// ---- 11_CNC/01_DUTs/02_ST/ST_CNC_Heidenhain_Exchange_Out_1.TcDUT
//-----------------------------------------------------------------------------------------
//
//                  				ST_CNC_Heidenhain_Exchange_Out
//
//								Structure Echange Magasin->CNC_Heidenhain 			
//-----------------------------------------------------------------------------------------
//
//Auteur: G.GOETZ (In agreement with ...)
//Création: 27.01.2026
//Dernière modification : 27.01.2026 (G.GOETZ)
//       			
//-----------------------------------------------------------------------------------------
//
//     							Liste des modifications  	
//
// 27.01.2026 (G.GOETZ) -> Création		
//-----------------------------------------------------------------------------------------

TYPE ST_CNC_Heidenhain_Exchange_Out_1 : // 16 Bytes -> Start at X0.0 / End at X15.7 (X0.0+15.7)
STRUCT
	
	(* Byte 0 *)
		boLife : BIT ; // Magazine Life bit -> X0.0
		boReserve01 : BIT ; // Reserve 01 -> X0.1
		boReserve02 : BIT ; // Reserve 02 -> X0.2
		boReserve03 : BIT ; // Reserve 03 -> X0.3
		boReserve04 : BIT ; // Reserve 04 -> X0.4
		boReserve05 : BIT ; // Reserve 05 -> X0.5
		boLoadingArmInPosition : BIT ; // Loading Arm in position in the CNC -> X0.6
		boNoFault : BIT ; // No Fault on the Magazine -> X0.7

	(* Byte 1 *)
		boReserve10 : BIT ; // Reserve 10 -> X1.0
		boReserve11 : BIT ; // Reserve 11 -> X1.1
		boReserve12 : BIT ; // Reserve 12 -> X1.2
		boReserve13 : BIT ; // Reserve 13 -> X1.3
		boReserve14 : BIT ; // Reserve 14 -> X1.4
		boReserve15 : BIT ; // Reserve 15 -> X1.5
		boReserve16 : BIT ; // Reserve 16 -> X1.6
		boDoorClosed : BIT ; // Magazine Door closed (operator) -> X1.7

	(* Byte 2 *)
		boReserve20 : BIT ; // Reserve 20 -> X2.0
		boReserve21 : BIT ; // Reserve 21 -> X2.1
		boReserve22 : BIT ; // Reserve 22 -> X2.2
		boReserve23 : BIT ; // Reserve 23 -> X2.3
		boReserve24 : BIT ; // Reserve 24 -> X2.4
		boReserve25 : BIT ; // Reserve 25 -> X2.5
		boReserve26 : BIT ; // Reserve 26 -> X2.6
		boReserve27 : BIT ; // Reserve 27 -> X2.7
	
	(* Byte 3 *)
		boReserve30 : BIT ; // Reserve 30 -> X3.0
		boReserve31 : BIT ; // Reserve 31 -> X3.1
		boReserve32 : BIT ; // Reserve 32 -> X3.2
		boReserve33 : BIT ; // Reserve 33 -> X3.3
		boReserve34 : BIT ; // Reserve 34 -> X3.4
		boReserve35 : BIT ; // Reserve 35 -> X3.5
		boReserve36 : BIT ; // Reserve 36 -> X3.6
		boReserve37 : BIT ; // Reserve 37 -> X3.7

	(* Byte 4 *)
		byoReserve40 : BYTE ; // Reserve 40 -> X4
	
	(* Byte 5 *)
		byoReserve50 : BYTE ; // Reserve 50 -> X5
	
	(* Byte 6 *)
		byoReserve60 : BYTE ; // Reserve 60 -> X6
	
	(* Byte 7 *)
		byoReserve70 : BYTE ; // Reserve 70 -> X7
	
	(* Byte 8 *)
		byoReserve80 : BYTE ; // Reserve 80 -> X8
	
	(* Byte 9 *)
		byoReserve90 : BYTE ; // Reserve 90 -> X9
		
	(* Byte 10 *)
		byoReserve100 : BYTE ; // Reserve 100 -> X10
	
	(* Byte 11 *)
		byoReserve110 : BYTE ; // Reserve 110 -> X11
	
	(* Byte 12 *)
		byoReserve120 : BYTE ; // Reserve 120 -> X12
	
	(* Byte 13 *)
		byoReserve130 : BYTE ; // Reserve 130 -> X13
	
	(* Byte 14 *)
		byoReserve140 : BYTE ; // Reserve 140 -> X14
	
	(* Byte 15 *)
		byoReserve150 : BYTE ; // Reserve 150 -> X15
	
END_STRUCT
END_TYPE

// ---- 11_CNC/01_DUTs/02_ST/ST_CNC_Heidenhain_Data.TcDUT
//-----------------------------------------------------------------------------------------
//
//                  				ST_CNC_Heidenhain_Data
//
//								Structure CNC_Heidenhain Data 			
//-----------------------------------------------------------------------------------------
//
//Auteur: G.GOETZ
//Création: 27.01.2026
//Dernière modification : 27.01.2026 (G.GOETZ)
//       			
//-----------------------------------------------------------------------------------------
//
//     							Liste des modifications  	
//
// 27.01.2026 (G.GOETZ) -> Création		
//-----------------------------------------------------------------------------------------

TYPE ST_CNC_Heidenhain_Data :
STRUCT

	(** ST **)	
		stCncMagazine : ST_CNC_Heidenhain_Exchange_In_1 ; // Structure Exchange CNC -> Magazine
		stMagazineCNC : ST_CNC_Heidenhain_Exchange_Out_1 ; // Structure Exchange Magzine -> CNC

END_STRUCT
END_TYPE

// ---- 11_CNC/01_DUTs/02_ST/ST_CNC_Fanuc_Exchange_In_1.TcDUT
//-----------------------------------------------------------------------------------------
//
//                  				ST_CNC_Fanuc_Exchange_In
//
//								Structure Echange CNC_Fanuc->Magasin 			
//-----------------------------------------------------------------------------------------
//
//Auteur: G.GOETZ (In agreement with J.SPÄTIG)
//Création: 27.01.2026
//Dernière modification : 27.01.2026 (G.GOETZ)
//       			
//-----------------------------------------------------------------------------------------
//
//     							Liste des modifications  	
//
// 27.01.2026 (G.GOETZ) -> Création		
//-----------------------------------------------------------------------------------------

TYPE ST_CNC_Fanuc_Exchange_In_1 : // 32 Bytes -> Start at X0.0 / End at X31.7 (X0.0+31.7)
STRUCT
	
	(* Byte 0 *)
		byi0 AT %I* : BYTE ; // Byte X0
			biLife : BIT ; // Life bit -> X0.0
			biToolAnticipation : BIT ; // Anticipation to prepare the next Tool -> X0.1
			biAllowedOpenIntermediateDoor : BIT ; // Allowed to open the Intermediate Door 02 -> X0.2
			biLoadUnloadRequest : BIT ; // Request to Load and Unload a Tool -> X0.3
			biLoadRequest : BIT ; // Request to only Load a Tool -> X0.4
			biUnloadRequest : BIT ; // Request to only Unload a Tool -> X0.5
			biLoadUnloadEnd : BIT ; // End of the Request -> X0.6
			biAllowedCloseIntermediateDoor : BIT ; // Allowed to close the Intermediate Door 07 -> X0.7

	(* Byte 1 *)
		byi1 AT %I* : BYTE ; // Byte X1
			biInCycle : BIT ; // CNC in Cycle -> X1.0
			biEvacuateArm : BIT ; // Request to evacuate the Changing Arm and close the Intermediate Door -> X1.1
			biReserve12 : BIT ; // Reserve 12 -> X1.2
				//biIntermediateDoorOpened : BIT ; // Intermediate magazine-cnc Door Opened -> X1.2
			biReserve13 : BIT ; // Reserve 13 -> X1.3
			biReserve14 : BIT ; // Reserve 14 -> X1.4
			biReserve15 : BIT ; // Reserve 15 -> X1.5
			biReserve16 : BIT ; // Reserve 16 -> X1.6
			biDoorClosed : BIT ; // CNC Door closed (operator) -> X1.7

	(* Byte 2 *)
		byi2 AT %I* : BYTE ; // Byte X2
			biEmergencyStop : BIT ; // Emergency Stop -> X2.0
			biPower : BIT ; // Power -> X2.1
			biAir : BIT ; // Air -> X2.2
			biShutdown : BIT ; // Shutdown -> X2.3
			biReserve24 : BIT ; // Reserve 24 -> X2.4
			biReserve25 : BIT ; // Reserve 25 -> X2.5
			biReserve26 : BIT ; // Reserve 26 -> X2.6
			biReserve27 : BIT ; // Reserve 27 -> X2.7
	
	(* Byte 3 *)
		byi3 AT %I* : BYTE ; // Byte X3
			biReserve30 : BIT ; // Reserve 30 -> X3.0
			biReserve31 : BIT ; // Reserve 31 -> X3.1
			biReserve32 : BIT ; // Reserve 32 -> X3.2
			biReserve33 : BIT ; // Reserve 33 -> X3.3
			biReserve34 : BIT ; // Reserve 34 -> X3.4
			biReserve35 : BIT ; // Reserve 35 -> X3.5
			biReserve36 : BIT ; // Reserve 36 -> X3.6
			biReserve37 : BIT ; // Reserve 37 -> X3.7

	(* Byte 4 *)
		byi4 AT %I* : BYTE ; // Byte X4
			biReserve40 : BIT ; // Reserve 40 -> X4.0
			biReserve41 : BIT ; // Reserve 41 -> X4.1
			biReserve42 : BIT ; // Reserve 42 -> X4.2
			biReserve43 : BIT ; // Reserve 43 -> X4.3
			biReserve44 : BIT ; // Reserve 44 -> X4.4
			biReserve45 : BIT ; // Reserve 45 -> X4.5
			biReserve46 : BIT ; // Reserve 46 -> X4.6
			biReserve47 : BIT ; // Reserve 47 -> X4.7

	(* Byte 5 *)
		byi5 AT %I* : BYTE ; // Byte X5
			biReserve50 : BIT ; // Reserve 50 -> X5.0
			biReserve51 : BIT ; // Reserve 51 -> X5.1
			biReserve52 : BIT ; // Reserve 52 -> X5.2
			biReserve53 : BIT ; // Reserve 53 -> X5.3
			biReserve54 : BIT ; // Reserve 54 -> X5.4
			biReserve55 : BIT ; // Reserve 55 -> X5.5
			biReserve56 : BIT ; // Reserve 56 -> X5.6
			biReserve57 : BIT ; // Reserve 57 -> X5.7

	(* Byte 6 *)
		byiSpindleToolType AT %I* : BYTE ; // Type of the Tool in CNC Spindle -> X6 (0=Unknow/1=Small/2=Big)
	
	(* Byte 7 *)
		byiToolToLoadType AT %I* : BYTE ; // Type of the Tool to Load in CNC Spindle -> X7 (0=Unknow/1=Small/2=Big)
	
	(* Byte 8-9 *)
		wiSpindleToolLocation AT %I* : WORD ; // Location of the Tool in CNC Spindle -> X8-9
	
	(* Byte 10-11 *)
		wiToolToLoadLocation AT %I* : WORD ; // Location of the Tool to Load in CNC Spindle -> X10-11

	(* Byte 12-13 *)
		wiPT100ArmorStatus AT %I* : WORD ; // PT100 probe in the electrical armor -> X12-13
	
	(* Byte 14-15 *)
		wiPT100ArmorValue AT %I* : WORD ; // PT100 probe in the electrical armor -> X14-15
		
	(* Byte 16 *)
		byiResevrve16 AT %I* : BYTE ; // Byte Reserve 16 -> X16
		
	(* Byte 17 *)
		byiResevrve17 AT %I* : BYTE ; // Byte Reserve 17 -> X17
		
	(* Byte 18 *)
		byiResevrve18 AT %I* : BYTE ; // Byte Reserve 18 -> X18
		
	(* Byte 19 *)
		byiResevrve19 AT %I* : BYTE ; // Byte Reserve 19 -> X19
		
	(* Byte 20 *)
		byiResevrve20 AT %I* : BYTE ; // Byte Reserve 20 -> X20
		
	(* Byte 21 *)
		byiResevrve21 AT %I* : BYTE ; // Byte Reserve 21 -> X21
		
	(* Byte 22 *)
		byiResevrve22 AT %I* : BYTE ; // Byte Reserve 22 -> X22
		
	(* Byte 23 *)
		byiResevrve23 AT %I* : BYTE ; // Byte Reserve 23 -> X23
		
	(* Byte 24 *)
		byiResevrve24 AT %I* : BYTE ; // Byte Reserve 24 -> X24
		
	(* Byte 25 *)
		byiResevrve25 AT %I* : BYTE ; // Byte Reserve 25 -> X20
		
	(* Byte 26 *)
		byiResevrve26 AT %I* : BYTE ; // Byte Reserve 26 -> X26
		
	(* Byte 27 *)
		byiResevrve27 AT %I* : BYTE ; // Byte Reserve 27 -> X27
		
	(* Byte 28 *)
		byiResevrve28 AT %I* : BYTE ; // Byte Reserve 28 -> X28
		
	(* Byte 29 *)
		byiResevrve29 AT %I* : BYTE ; // Byte Reserve 29 -> X29
		
	(* Byte 30 *)
		byiResevrve30 AT %I* : BYTE ; // Byte Reserve 30 -> X30
		
	(* Byte 31 *)
		byiResevrve31 AT %I* : BYTE ; // Byte Reserve 31 -> X31
		
END_STRUCT
END_TYPE

// ---- 11_CNC/01_DUTs/02_ST/ST_CNC_Fanuc_Exchange_Out_1.TcDUT
//-----------------------------------------------------------------------------------------
//
//                  				ST_CNC_Fanuc_Exchange_Out
//
//								Structure Echange Magasin->CNC_Fanuc 			
//-----------------------------------------------------------------------------------------
//
//Auteur: G.GOETZ (In agreement with J.SPÄTIG)
//Création: 27.01.2026
//Dernière modification : 27.01.2026 (G.GOETZ)
//       			
//-----------------------------------------------------------------------------------------
//
//     							Liste des modifications  	
//
// 27.01.2026 (G.GOETZ) -> Création		
//-----------------------------------------------------------------------------------------

TYPE ST_CNC_Fanuc_Exchange_Out_1 : // 32 Bytes -> Start at X0.0 / End at X31.7 (X0.0+31.7)
STRUCT
	
	(* Byte 0 *)
		byo0 AT %Q* : BYTE ; // Byte X0
			boLife : BIT ; // Magazine Life bit -> X0.0
			boToolAnticipated : BIT ; // Next tool is prepared/anticipated -> X0.1
			boReserve02 : BIT ; // Reserve 02 -> X0.2
			boReserve03 : BIT ; // Reserve 03 -> X0.3
			boReserve04 : BIT ; // Reserve 04 -> X0.4
			boReserve05 : BIT ; // Reserve 05 -> X0.5
			boArmInCncPosition : BIT ; // Loading Arm in position in the CNC -> X0.6
			boNoFault : BIT ; // No Fault on the Magazine -> X0.7

	(* Byte 1 *)
		byo1 AT %Q* : BYTE ; // Byte X1
			boArmOutOfCncArea : BIT ; // Changing Arm out of Cnc area -> X1.0
			boOpenManipulatorGripper : BIT ; // Open the manipulator gripper -> X1.1
			boAirBlowIntermediateDoor : BIT ; // Air blow of the Intermediate Door -> X1.2
			boIntermediateDoorOpen : BIT ; // Intermediate Door is open -> X1.3
			boIntermediateDoorClose : BIT ; // Intermediate Door is close -> X1.4
			boReserve15 : BIT ; // Reserve 15 -> X1.5
			boReserve16 : BIT ; // Reserve 16 -> X1.6
			boReserve17 : BIT ; // Reserve 17 -> X1.7
			
	(* Byte 2 *)
		byo2 AT %Q* : BYTE ; // Byte X2
			boReserve20 : BIT ; // Reserve 20 -> X2.0
			boReserve21 : BIT ; // Reserve 21 -> X2.1
			boReserve22 : BIT ; // Reserve 22 -> X2.2
			boReserve23 : BIT ; // Reserve 23 -> X2.3
			boReserve24 : BIT ; // Reserve 24 -> X2.4
			boReserve25 : BIT ; // Reserve 25 -> X2.5
			boReserve26 : BIT ; // Reserve 26 -> X2.6
			boReserve27 : BIT ; // Reserve 27 -> X2.7
	
	(* Byte 3 *)
		byo3 AT %Q* : BYTE ; // Byte X3
			boReserve30 : BIT ; // Reserve 30 -> X3.0
			boReserve31 : BIT ; // Reserve 31 -> X3.1
			boReserve32 : BIT ; // Reserve 32 -> X3.2
			boReserve33 : BIT ; // Reserve 33 -> X3.3
			boReserve34 : BIT ; // Reserve 34 -> X3.4
			boReserve35 : BIT ; // Reserve 35 -> X3.5
			boReserve36 : BIT ; // Reserve 36 -> X3.6
			boReserve37 : BIT ; // Reserve 37 -> X3.7

	(* Byte 4 *)
		byo4 AT %Q* : BYTE ; // Byte X4
			boReserve40 : BIT ; // Reserve 40 -> X4.0
			boReserve41 : BIT ; // Reserve 41 -> X4.1
			boReserve42 : BIT ; // Reserve 42 -> X4.2
			boReserve43 : BIT ; // Reserve 43 -> X4.3
			boReserve44 : BIT ; // Reserve 44 -> X4.4
			boReserve45 : BIT ; // Reserve 45 -> X4.5
			boReserve46 : BIT ; // Reserve 46 -> X4.6
			boReserve47 : BIT ; // Reserve 47 -> X4.7

	(* Byte 5 *)
		byo5 AT %Q* : BYTE ; // Byte X5
			boReserve50 : BIT ; // Reserve 50 -> X5.0
			boReserve51 : BIT ; // Reserve 51 -> X5.1
			boReserve52 : BIT ; // Reserve 52 -> X5.2
			boReserve53 : BIT ; // Reserve 53 -> X5.3
			boReserve54 : BIT ; // Reserve 54 -> X5.4
			boReserve55 : BIT ; // Reserve 55 -> X5.5
			boReserve56 : BIT ; // Reserve 56 -> X5.6
			boReserve57 : BIT ; // Reserve 57 -> X5.7

	(* Byte 6 *)
		byoResevrve6 AT %Q* : BYTE ; // Byte Reserve 6 -> X6

	(* Byte 7 *)
		byoResevrve7 AT %Q* : BYTE ; // Byte Reserve 7 -> X7

	(* Byte 8-9 *)
		woReserve8 AT %Q* : WORD ; // Word Reserve 8 -> X8-9
	
	(* Byte 10-11 *)
		woReserve10 AT %Q* : WORD ; // Word Reserve 10 -> X10-11

	(* Byte 12-13 *)
		woResevrve12 AT %Q* : WORD ; // Word Reserve 12 -> X12-X13
		
	(* Byte 14-15 *)
		woResevrve14 AT %Q* : WORD ; // Word Reserve 14 -> X14-X15
		
	(* Byte 16 *)
		byoResevrve16 AT %Q* : BYTE ; // Byte Reserve 16 -> X16
		
	(* Byte 17 *)
		byoResevrve17 AT %Q* : BYTE ; // Byte Reserve 17 -> X17
		
	(* Byte 18 *)
		byoResevrve18 AT %Q* : BYTE ; // Byte Reserve 18 -> X18
		
	(* Byte 19 *)
		byoResevrve19 AT %Q* : BYTE ; // Byte Reserve 19 -> X19
		
	(* Byte 20 *)
		byoResevrve20 AT %Q* : BYTE ; // Byte Reserve 20 -> X20
		
	(* Byte 21 *)
		byoResevrve21 AT %Q* : BYTE ; // Byte Reserve 21 -> X21
		
	(* Byte 22 *)
		byoResevrve22 AT %Q* : BYTE ; // Byte Reserve 22 -> X22
		
	(* Byte 23 *)
		byoResevrve23 AT %Q* : BYTE ; // Byte Reserve 23 -> X23
		
	(* Byte 24 *)
		byoResevrve24 AT %Q* : BYTE ; // Byte Reserve 24 -> X24
		
	(* Byte 25 *)
		byoResevrve25 AT %Q* : BYTE ; // Byte Reserve 25 -> X20
		
	(* Byte 26 *)
		byoResevrve26 AT %Q* : BYTE ; // Byte Reserve 26 -> X26
		
	(* Byte 27 *)
		byoResevrve27 AT %Q* : BYTE ; // Byte Reserve 27 -> X27
		
	(* Byte 28 *)
		byoResevrve28 AT %Q* : BYTE ; // Byte Reserve 28 -> X28
		
	(* Byte 29 *)
		byoResevrve29 AT %Q* : BYTE ; // Byte Reserve 29 -> X29
		
	(* Byte 30 *)
		byoResevrve30 AT %Q* : BYTE ; // Byte Reserve 30 -> X30
		
	(* Byte 31 *)
		byoResevrve31 AT %Q* : BYTE ; // Byte Reserve 31 -> X31
		
END_STRUCT
END_TYPE

// ---- 11_CNC/01_DUTs/02_ST/ST_Spindle.TcDUT
//-----------------------------------------------------------------------------------------
//
//                  				ST_Spindle
//
//								Structure Broche 			
//-----------------------------------------------------------------------------------------
//
//Auteur: G.GOETZ
//Création: 27.01.2026
//Dernière modification : 27.01.2026 (G.GOETZ)
//       			
//-----------------------------------------------------------------------------------------
//
//     							Liste des modifications  	
//
// 27.01.2026 (G.GOETZ) -> Création		
//-----------------------------------------------------------------------------------------

TYPE ST_Spindle :
STRUCT
	
	(** ST **)
		stLocationMemory : ST_Tool_location ; // Tool_Location structure
		
	(** PROCESS INT **)
		iAbsLocationNumberMemory : INT := 0 ; // Memory -> Number of the location in the Magazine
		iRelLocationNumberMemory : INT ; // Memory -> Number of the location in relative in the Magazine
		
	(** PROCESS FLAG **)
		bToolPresenceMemory : BOOL ; // Memory -> Tool Presence in the Manipulator
	
END_STRUCT
END_TYPE

// ---- 12_Focas/01_DUTs/02_ST/St_Write_Focas.TcDUT
//-----------------------------------------------------------------------------------------
//
//                  				ST_Write_Focas
//
//							Structure pour écriture Focas			
//-----------------------------------------------------------------------------------------
//
//Auteur: G.GOETZ (inspired by S.MANTZER)
//Création: 19.02.2026
//Dernière modification : 19.02.2026 (G.GOETZ)
//       			
//-----------------------------------------------------------------------------------------
//
//     							Liste des modifications  	
//
// 19.02.2026 (G.GOETZ) -> Création		
//-----------------------------------------------------------------------------------------

TYPE St_Write_Focas :
STRUCT
	
	(** ARRAY **)
		aTabValeur : ARRAY [0..499]	OF BYTE ; // Récupération des valeurs à écrire
	
	(** UINT **)			
		uiTypePMC : UINT ; // Type de variable à écrire dans le PMC
		uiTypeData : UINT ; // Type de donnée à lire (0 = byte, 1 = Word, 2 = Long, 4 = 32-bit floating-point type(30i-B Series/0i-F/PMi-A only), 5 = 64-bit floating-point type(30i-B Series/0i-F/PMi-A only) 
		uiBitLect : UINT ; // Numéro du bit à lire dans un word dans le PMC
		uiGrandType : UINT ; // Grandeur du block de donnée à lire Exemple : data_type is 0(byte type) : length = 8 + N			
		uiPMCAdr1 : UINT ; // Adresse de début de la donnée à lire
		uiPMCAdr2 : UINT ; // Adresse de fin de la donnée à lire
						
END_STRUCT
END_TYPE

// ---- 12_Focas/01_DUTs/02_ST/ST_Focas_To_Magazine.TcDUT
//-----------------------------------------------------------------------------------------
//
//                  				ST_Focas_To_Magazine
//
//							Structure échanges Focas vers Magasin			
//-----------------------------------------------------------------------------------------
//
//Auteur: G.GOETZ
//Création: 20.01.2026
//Dernière modification : 20.01.2026 (G.GOETZ)
//       			
//-----------------------------------------------------------------------------------------
//
//     							Liste des modifications  	
//
// 20.01.2026 (G.GOETZ) -> Création		
//-----------------------------------------------------------------------------------------

TYPE ST_Focas_To_Magazine :
STRUCT
	
	(** ARRAY ST **)
	aToolParamIn : ARRAY[1..GV_Tool_Magazine.iMaxAbsLocation] OF ST_Tool_Parameters ; // Tool_Parameters structure
	aToolNameIn : ARRAY[1..GV_Tool_Magazine.iMaxAbsLocation] OF ST_Tool_Name ; // Tool_Name structure
	
	(** PROCESS FLAG **)
	bRefreshIn : BOOL ; // Refresh Exchange
	
END_STRUCT
END_TYPE

// ---- 12_Focas/01_DUTs/02_ST/St_Read_Focas.TcDUT
//-----------------------------------------------------------------------------------------
//
//                  				ST_Read_Focas
//
//							Structure pour lecture Focas			
//-----------------------------------------------------------------------------------------
//
//Auteur: G.GOETZ (inspired by S.MANTZER)
//Création: 19.02.2026
//Dernière modification : 19.02.2026 (G.GOETZ)
//       			
//-----------------------------------------------------------------------------------------
//
//     							Liste des modifications  	
//
// 19.02.2026 (G.GOETZ) -> Création		
//-----------------------------------------------------------------------------------------


TYPE St_Read_Focas :
	{attribute 'packmode' := 2 }
STRUCT
	
	(** ARRAY **)
		aTabValeur : ARRAY [0..499]	OF BYTE ; // Récupération des valeurs à écrire
	
	(** UINT **)			
		uiTypePMC : UINT ; // Type de variable à écrire dans le PMC
		uiTypeData : UINT ; // Type de donnée à lire (0 = byte, 1 = Word, 2 = Long, 4 = 32-bit floating-point type(30i-B Series/0i-F/PMi-A only), 5 = 64-bit floating-point type(30i-B Series/0i-F/PMi-A only) 
		uiBitLect : UINT ; // Numéro du bit à lire dans un word dans le PMC
		uiGrandType : UINT ; // Grandeur du block de donnée à lire Exemple : data_type is 0(byte type) : length = 8 + N			
		uiPMCAdr1 : UINT ; // Adresse de début de la donnée à lire
		uiPMCAdr2 : UINT ; // Adresse de fin de la donnée à lire

END_STRUCT
END_TYPE

// ---- 12_Focas/01_DUTs/02_ST/ST_Magazine_To_Focas.TcDUT
//-----------------------------------------------------------------------------------------
//
//                  				ST_Magazine_To_Focas
//
//							Structure échanges Magasin vers Focas			
//-----------------------------------------------------------------------------------------
//
//Auteur: G.GOETZ
//Création: 20.01.2026
//Dernière modification : 20.01.2026 (G.GOETZ)
//       			
//-----------------------------------------------------------------------------------------
//
//     							Liste des modifications  	
//
// 20.01.2026 (G.GOETZ) -> Création		
//-----------------------------------------------------------------------------------------

TYPE ST_Magazine_To_Focas :
STRUCT
		
	(** ARRAY ST **)
	aToolParamOut : ARRAY[1..GV_Tool_Magazine.iMaxAbsLocation] OF ST_Tool_Parameters ; // Tool_Parameters structure
	aToolNameOut : ARRAY[1..GV_Tool_Magazine.iMaxAbsLocation] OF ST_Tool_Name ; // Tool_Name structure
	
	(** PROCESS FLAG **)
	bRefreshOut : BOOL ; // Refresh Exchange
	
END_STRUCT
END_TYPE

// ---- 13_HMI/01_DUTs/01_ENUM/ENUM_User_Level.TcDUT
{attribute 'qualified_only'}
{attribute 'strict'}

//-----------------------------------------------------------------------------------------
//
//                  				ENUM_User_Level
//
//							Enumération des niveaux d'utilisateurs			
//-----------------------------------------------------------------------------------------
//
//Auteur: G.GOETZ
//Création: 04.03.2026
//Dernière modification : 04.03.2026 (G.GOETZ)
//       			
//-----------------------------------------------------------------------------------------
//
//     							Liste des modifications  	
//
// 04.03.2026 (G.GOETZ) -> Création		
//-----------------------------------------------------------------------------------------

TYPE ENUM_User_Level :
(
	None := 0 ,
	Admin := 1 ,
	Maintenance := 2 ,
	Operator := 3 
);
END_TYPE

// ---- 13_HMI/01_DUTs/02_ST/ST_HMI_Axes.TcDUT
//-----------------------------------------------------------------------------------------
//
//                  				ST_HMI_Axes
//
//								Structure Axes HMI			
//-----------------------------------------------------------------------------------------
//
//Auteur: G.GOETZ
//Création: 20.02.2026
//Dernière modification : 20.02.2026 (G.GOETZ)
//       			
//-----------------------------------------------------------------------------------------
//
//     							Liste des modifications  	
//
// 20.02.2026 (G.GOETZ) -> Création		
//-----------------------------------------------------------------------------------------

TYPE ST_HMI_Axes :
STRUCT
	
	(** SETUP LREAL **)
		lrVelocityPourcent : LREAL ; // Velocity in Pourcent

	(** SETUP INT **)
		iVelocityPourcent : INT ; // Velocity in Pourcent

	(** SETUP FLAG **)
		bButtonChoiceAxisX : BOOL ; // Button Axis Choice X
			rtButtonChoiceAxisX : R_Trig ; // Trigger for Button Axis Choice X
		bButtonChoiceAxisY : BOOL ; // Button Axis Choice Y
			rtButtonChoiceAxisY : R_Trig ; // Trigger for Button Axis Choice Y
		bButtonChoiceAxisZ : BOOL ; // Button Axis Choice Z
			rtButtonChoiceAxisZ : R_Trig ; // Trigger for Button Axis Choice Z
		bButtonChoiceAxisArm : BOOL ; // Button Axis Choice Arm
			rtButtonChoiceAxisArm : R_Trig ; // Trigger for Button Axis Choice Arm	
		
		bButtonPlus : BOOL ; // Button Plus
			rtButtonPlus : R_Trig ; // Trigger for Button Plus
		bButtonMinus : BOOL ; // Button Minus
			rtButtonMinus : R_Trig ; // Trigger for Button Minus

		bButtonChoiceReferencingX : BOOL ; // Button Axis Referencing X
			rtButtonChoiceReferencingX : R_Trig ; // Trigger for Button Axis Referencing X
		bButtonChoiceReferencingY : BOOL ; // Button Axis Referencing Y
			rtButtonChoiceReferencingY : R_Trig ; // Trigger for Button Axis Referencing Y
		bButtonChoiceReferencingZ : BOOL ; // Button Axis Referencing Z
			rtButtonChoiceReferencingZ : R_Trig ; // Trigger for Button Axis Referencing Z
		bButtonChoiceReferencingArm : BOOL ; // Button Axis Referencing Arm
			rtButtonChoiceReferencingArm : R_Trig ; // Trigger for Button Axis Referencing Arm	
	
		bButtonReferencingAxis : BOOL ; // Button Referencing
			rtButtonReferencingAxis : R_Trig ; // Trigger for Button Referncing	
	
		bButtonMinSofltLimit : BOOL ; // Button Enable/Disable Min Soft Limit (for referencing)
			rtButtonMinSofltLimit : R_Trig ; // Trigger for Buttonnable/Disable Min Soft Limit (for referencing)
		bButtonMaxSofltLimit : BOOL ; // Button Enable/Disable Max Soft Limit (for referencing)
			rtButtonMaxSofltLimit : R_Trig ; // Trigger for Buttonnable/Disable Max Soft Limit (for referencing)
			
	(** PROCESS STRING **)
		sAxisXActPos : STRING ; // Actual Position of the Axis X
			lrAxisXActPos : LREAL ; // Actual Position of the Axis X
		sAxisXActVelo : STRING ; // Actual Velocity of the Axis X
			lrAxisXActVelo : LREAL ; // Actual Velocity of the Axis X
		sAxisYActPos : STRING ; // Actual Position of the Axis Y
			lrAxisYActPos : LREAL ; // Actual Position of the Axis Y
		sAxisYActVelo : STRING ; // Actual Velocity of the Axis Y
			lrAxisYActVelo : LREAL ; // Actual Velocity of the Axis Y
		sAxisZActPos : STRING ; // Actual Position of the Axis Z
			lrAxisZActPos : LREAL ; // Actual Position of the Axis Z
		sAxisZActVelo : STRING ; // Actual Velocity of the Axis Z
			lrAxisZActVelo : LREAL ; // Actual Velocity of the Axis Z
		sAxisArmActPos : STRING ; // Actual Position of the Axis Arm
			lrAxisArmActPos : LREAL ; // Actual Position of the Axis Arm
		sAxisArmActVelo : STRING ; // Actual Velocity of the Axis Arm
			lrAxisArmActVelo : LREAL ; // Actual Velocity of the Axis Arm
			
		sRefrencingActPos : STRING ; // Actual Position of the Axis choice for the referncing
			lrRefrencingActPos : LREAL ; // Actual Position of the Axis choice for the referncing
		
END_STRUCT
END_TYPE

// ---- 13_HMI/01_DUTs/02_ST/ST_HMI_Backup.TcDUT
//-----------------------------------------------------------------------------------------
//
//                  				ST_HMI_Backup
//
//								Structure Backup HMI			
//-----------------------------------------------------------------------------------------
//
//Auteur: G.GOETZ
//Création: 11.03.2026
//Dernière modification : 11.03.2026 (G.GOETZ)
//       			
//-----------------------------------------------------------------------------------------
//
//     							Liste des modifications  	
//
// 11.03.2026 (G.GOETZ) -> Création		
//-----------------------------------------------------------------------------------------

TYPE ST_HMI_Backup :
STRUCT
	
	(** FLAG + R_Trig **)
		bButtonProject : BOOL ; // Button for Backup Project
			rtButtonProject : R_TRIG ; // Trigger for Backup Project	
	
		bButtonInitData : BOOL ; // Button for Init data of the Export/Import Array
			rtButtonInitData : R_TRIG ; // Trigger for Init data of the Export/Import Array
		bButtonExportData : BOOL ; // Button for Export data
			rtButtonExportData : R_TRIG ; // Trigger for Export data
		bButtonImportData : BOOL ; // Button for Import data
			rtButtonImportData : R_TRIG ; // Trigger for Import data
			
		bButtonExportAlarms : BOOL ; // Button for Export alarms
			rtButtonExportAlarms : R_TRIG ; // Trigger for Export alarms
		bButtonExportMessages : BOOL ; // Button for Export messages
			rtButtonExportMessages : R_TRIG ; // Trigger for Export messages
		
END_STRUCT
END_TYPE

// ---- 13_HMI/01_DUTs/02_ST/ST_HMI_Cycle.TcDUT
//-----------------------------------------------------------------------------------------
//
//                  				ST_HMI_Cycle
//
//								Structure Cycle HMI			
//-----------------------------------------------------------------------------------------
//
//Auteur: G.GOETZ
//Création: 05.03.2026
//Dernière modification : 05.03.2026 (G.GOETZ)
//       			
//-----------------------------------------------------------------------------------------
//
//     							Liste des modifications  	
//
// 05.03.2026 (G.GOETZ) -> Création		
//-----------------------------------------------------------------------------------------

TYPE ST_HMI_Cycle :
STRUCT

	(** STRING **)
		sCurrentCycle : STRING(100) ;
		//sCurrentCycleStep : STRING(50) ;

	(** FLAG + R_Trig **)
		bButtonStartStop : BOOL ; // Button for Start/Stop Cycle
			rtButtonStartStop : R_TRIG ; // Trigger for Start/Stop Cycle
		bButtonStart : BOOL ; // Button for Start Cycle
			rtButtonStart : R_TRIG ; // Trigger for Start Cycle
		bButtonStop : BOOL ; // Button for Stop Cycle
			rtButtonStop : R_TRIG ; // Trigger for Stop Cycle

END_STRUCT
END_TYPE

// ---- 13_HMI/01_DUTs/02_ST/ST_HMI_Cyltronic.TcDUT
//-----------------------------------------------------------------------------------------
//
//                  				ST_HMI_Cyltronic
//
//								Structure Cyltronic HMI			
//-----------------------------------------------------------------------------------------
//
//Auteur: G.GOETZ
//Création: 05.03.2026
//Dernière modification : 05.03.2026 (G.GOETZ)
//       			
//-----------------------------------------------------------------------------------------
//
//     							Liste des modifications  	
//
// 05.03.2026 (G.GOETZ) -> Création		
//-----------------------------------------------------------------------------------------

TYPE ST_HMI_Cyltronic :
STRUCT
	
	(** PROCESS FLAG + R_TRIG **)
		bButtonMoveWork : BOOL ; // Button for move to Work Position
			rtButtonMoveWork : R_Trig ; // Trigger for move to Work Position
		bButtonMoveRest : BOOL ; // Button for move to Rest Position
			rtButtonMoveRest : R_Trig ; // Trigger for move to Rest Position
				
END_STRUCT
END_TYPE

// ---- 13_HMI/01_DUTs/02_ST/ST_HMI_Doors.TcDUT
//-----------------------------------------------------------------------------------------
//
//                  				ST_HMI_Doors
//
//								Structure portes HMI			
//-----------------------------------------------------------------------------------------
//
//Auteur: G.GOETZ
//Création: 20.02.2026
//Dernière modification : 20.02.2026 (G.GOETZ)
//       			
//-----------------------------------------------------------------------------------------
//
//     							Liste des modifications  	
//
// 20.02.2026 (G.GOETZ) -> Création		
//-----------------------------------------------------------------------------------------

TYPE ST_HMI_Doors :
STRUCT

	(** SETUP FLAG **)
		bDoorUnlockForce : BOOL ; // Door unlocking force

END_STRUCT
END_TYPE

// ---- 13_HMI/01_DUTs/02_ST/ST_HMI_Footer.TcDUT
//-----------------------------------------------------------------------------------------
//
//                  				ST_HMI_Footer
//
//							Structure datas pied de page HMI 			
//-----------------------------------------------------------------------------------------
//
//Auteur: G.GOETZ
//Création: 21.01.2026
//Dernière modification : 21.01.2026 (G.GOETZ)
//       			
//-----------------------------------------------------------------------------------------
//
//     							Liste des modifications  	
//
// 21.01.2026 (G.GOETZ) -> Création		
//-----------------------------------------------------------------------------------------

TYPE ST_HMI_Footer :
STRUCT
	
	(** SETUP INT **)
		ix1 : INT ; // ?
	
	(** SETUP FLAG **)
		bx1 : BOOL ; // ?

	(** PROCESS INT **)
		iy1 : INT ; // ?
	
	(** PROCESS FLAG **)
		by1 : BOOL ; // ?
	
END_STRUCT
END_TYPE

// ---- 13_HMI/01_DUTs/02_ST/ST_HMI_Header.TcDUT
//-----------------------------------------------------------------------------------------
//
//                  				ST_HMI_Header
//
//							Structure datas en-tête HMI 			
//-----------------------------------------------------------------------------------------
//
//Auteur: G.GOETZ
//Création: 21.01.2026
//Dernière modification : 21.01.2026 (G.GOETZ)
//       			
//-----------------------------------------------------------------------------------------
//
//     							Liste des modifications  	
//
// 21.01.2026 (G.GOETZ) -> Création		
//-----------------------------------------------------------------------------------------

TYPE ST_HMI_Header :
STRUCT
	
	(** SETUP INT **)
		ix1 : INT ; // ?
	
	(** SETUP FLAG **)
		bx1 : BOOL ; // ?

	(** PROCESS INT **)
		iy1 : INT ; // ?
	
	(** PROCESS FLAG **)
		by1 : BOOL ; // ?
	
END_STRUCT
END_TYPE

// ---- 13_HMI/01_DUTs/02_ST/ST_HMI_Lamps_Lights.TcDUT
//-----------------------------------------------------------------------------------------
//
//                  			ST_HMI_Lamps_Lights
//
//							Structure voyants et lumières HMI 			
//-----------------------------------------------------------------------------------------
//
//Auteur: G.GOETZ (inspired by S.MANTZER)
//Création: 13.01.2026
//Dernière modification : 13.01.2026 (G.GOETZ)
//       			
//-----------------------------------------------------------------------------------------
//
//     							Liste des modifications  	
//
// 13.01.2026 (G.GOETZ) -> Création		
//-----------------------------------------------------------------------------------------

TYPE ST_HMI_Lamps_Lights :
STRUCT
	
	(** SETUP INT **)
		iLightsTimer : INT ; // Value of the lights timer
	
	(** SETUP FLAG **)
		bLightsWithTimer : BOOL ; // Lights work with timer
	
	(** PROCESS FLAG **)
		bLightsButton : BOOL ; // Button for lights
		
		bLampInit : BOOL ; // Lamp for Init
		bLampAuto : BOOL ; // Lamp for Auto
		bLampManu : BOOL ; // Lamp for Manu
		bLampAck : BOOL ; // Lamp for acknowledgement
		
		bLampStartCycle : BOOL ; // Lamp for Start Cyle
		bLampStopCycle : BOOL ; // Lamp for Stop

		bLampManuManipGripperCloseEnable : BOOL ; // Lamp for Close Manipulator Gripper Enable
		bLampManuManipGripperOpenEnable : BOOL ; // Lamp for Open Manipulator Gripper Enable
		
		bLampManuCyltronicRestEnable : BOOL ; // Lamp for move to Rest cyltronic Enable
		bLampManuCyltronicWorkEnable : BOOL ; // Lamp for move to Work cyltronic Enable
		
		bLampAxisXOperationnal : BOOL ; // Lamp for Axis X Operationnal
		bLampAxisYOperationnal : BOOL ; // Lamp for Axis X Operationnal
		bLampAxisZOperationnal : BOOL ; // Lamp for Axis X Operationnal
		bLampAxisArmOperationnal : BOOL ; // Lamp for Axis X Operationnal
		
		bLampJogAxisX : BOOL ; // Lamp for Axis X choice in Jog
		bLampJogAxisY : BOOL ; // Lamp for Axis Y choice in Jog
		bLampJogAxisZ : BOOL ; // Lamp for Axis Z choice in Jog
		bLampJogAxisArm : BOOL ; // Lamp for Axis Arm choice in Jog
		
		bLampRefAxisX : BOOL ; // Lamp for Axis X referencing
		bLampRefAxisY : BOOL ; // Lamp for Axis Y referencing
		bLampRefAxisZ : BOOL ; // Lamp for Axis Z referencing
		bLampRefAxisArm : BOOL ; // Lamp for Axis Arm referencing
		
		bLampEnMinSoftPosLimit : BOOL ; // Lamp for Min Soft Limit Enable/Disable of the Axis referencing
		bLampEnMaxSoftPosLimit : BOOL ; // Lamp for Max Soft Limit Enable/Disable of the Axis referencing

		bLampBackupProjectEnable : BOOL ; // Lamp for Backup Project Enable
		bLampDataInitEnable : BOOL ; // Lamp for Init data Enable		
		bLampDataExportEnable : BOOL ; // Lamp for Export data Enable
		bLampDataImportEnable : BOOL ; // Lamp for Import data Enable
		bLampAlarmsExportEnable : BOOL ; // Lamp for Export alarms Enable
		bLampMessagesExportEnable : BOOL ; // Lamp for Export messages Enable
		
		bLampProject : BOOL ; // Lamp for project backup in progress
		bLampDataInit : BOOL ; // Lamp for Init data in progress
		bLampDataExport : BOOL ; // Lamp for Export data in progress
		bLampDataImport : BOOL ; // Lamp for Import data in progress
		
		bLampTeachLocationEnable : BOOL ; // Lamp for Teach Location Enable
		bLampTeachRackEnable : BOOL ; // Lamp for Teach Rack Enable
		bLampTeachAllTopEnable : BOOL ; // Lamp for Teach AllTop Enable
		bLampTeachAllBottomEnable : BOOL ; // Lamp for Teach AllBottom Enable
		bLampTeachPositionsEnable : BOOL ; // Lamp for Teach Positions Enable
		
		bLampRebootEnable : BOOL ; // Lamp for Reboot Enable
		bLampShutdownEnable : BOOL ; // Lamp for Shutdown Enable
		
		bLampSettingsSaveEnable : BOOL ; // Lamp for Save Settings Enable
		
END_STRUCT
END_TYPE

// ---- 13_HMI/01_DUTs/02_ST/ST_HMI_Magazine_Check.TcDUT
//-----------------------------------------------------------------------------------------
//
//                  			ST_HMI_Magazine_Check
//
//						Structure datas pour le check du magasin			
//-----------------------------------------------------------------------------------------
//
//Auteur: G.GOETZ
//Création: 17.02.2026
//Dernière modification : 17.02.2026 (G.GOETZ)
//       			
//-----------------------------------------------------------------------------------------
//
//     							Liste des modifications  	
//
// 17.02.2026 (G.GOETZ) -> Création		
//-----------------------------------------------------------------------------------------

TYPE ST_HMI_Magazine_Check :
STRUCT

	(** SETUP TIME **)
		tTimeoutOne : TIME ; // Value of the timeout for the check One
		tTimeoutFull : TIME ; // Value of the timeout for the check Full
		
	(** SETUP LREAL **)
		lrToolDistance : LREAL ; // Theoretical distance in mm for tool presence
		lrToolDistanceTolerance : LREAL ; // Tolerance in distance in mm for tool presence
		
	(** SETUP INT **)
		iTimeoutOne : INT ; // Value of the timeout for the check One
		iTimeoutFull : INT ; // Value of the timeout for the check Full
		iCheckCycleType : INT ; // Type of the Check Magazine cycle
		
	(** SETUP FLAG **)
		bCheckManipulatorLocation : BOOL ; // Check or not Manipulator Location when CheckMagazineOne
		bCheckArmGripper1Location : BOOL ; // Check or not Arm Gripper 1 Location when CheckMagazineOne
		bCheckArmGripper2Location : BOOL ; // Check or not Arm Gripper 2 Location when CheckMagazineOne
		bCheckSpindleLocation : BOOL ; // Check or not Spindle Location when CheckMagazineOne
		
END_STRUCT
END_TYPE

// ---- 13_HMI/01_DUTs/02_ST/ST_HMI_Magazine_Settings.TcDUT
//-----------------------------------------------------------------------------------------
//
//                  			ST_HMI_Magazine_Settings
//
//					Structure datas pour la configuration du magasin			
//-----------------------------------------------------------------------------------------
//
//Auteur: G.GOETZ
//Création: 17.03.2026
//Dernière modification : 17.03.2026 (G.GOETZ)
//       			
//-----------------------------------------------------------------------------------------
//
//     							Liste des modifications  	
//
// 17.03.2026 (G.GOETZ) -> Création		
//-----------------------------------------------------------------------------------------

TYPE ST_HMI_Magazine_Settings :
STRUCT
	
	(** SETUP LREAL **)
		(* Top *)
			lrZAbsCompensationLocationTop : LREAL ; // Z compensation total for the locations at the top in mm
	
			lrXLocationOffsetTop : LREAL ; // X Offset between location at the top of the Magazine
			lrYLocationOffsetTop : LREAL ; // Y Offset between location at the top of the Magazine
			lrZLocationOffsetTop : LREAL ; // Z Offset between location at the top of the Magazine
			
			lrXFirstLocationTop : LREAL ; // X of the first location at the top of the Magazine
			lrYLocationTop : LREAL ; // Y of the Location at the top of the Magazine
			lrZLowestRackTop : LREAL ; // Z of the lowest rack at the top of the Magazine
			
		(* Bottom *)
			lrZAbsCompensationLocationBottom : LREAL ; // Z compensation total for the locations at the bottom in mm
			
			lrXLocationOffsetBottom : LREAL ; // X Offset between location at the bottom of the Magazine
			lrYLocationOffsetBottom : LREAL ; // Y Offset between location at the bottom of the Magazine
			lrZLocationOffsetBottom : LREAL ; // Z Offset between location at the bottom of the Magazine
			
			lrXFirstLocationBottom : LREAL ; // X of the first location at the bottom of the Magazine
			lrYLocationBottom : LREAL ; // Y of the Location at the bottom of the Magazine
			lrZLowestRackBottom : LREAL ; // Z of the first lowest at the bottom of the Magazine
	
	
		lrYOffsetFrontLocation : LREAL ; // Y Offset to be in front of the Y coordinate of the location
		lrZOffsetAboveLocation : LREAL ; // Z Offset to be above of the Z coordinate of the location

		lrZOffsetAboveArmGripper1 : LREAL ; // Z Offset to be above the Z coordinate of the changing arm gripper 1 when in tansfer position
		lrZOffsetAboveArmGripper2 : LREAL ; // Z Offset to be above the Z coordinate of the changing arm gripper 2 when in tansfer position
		
		lrZOffsetToolCheck : LREAL ; // Z Offset above the tool for the check
		lrYOffsetToolCheck : LREAL ; // Y Offset in foront of the tool for the check
	
	(** SETUP REAL **)
		rZBrakeTimer : REAL ; // Timer before brake axis Z 
	
	(** SETUP INT **)
		iMaxRelRackLocationTop : INT ; // Max Location in a Rack in relative at the top of the Magazine
		iMaxRelRackLocationBottom : INT ; // Max Location in a Rack in relative at the bottom of the Magazine
		iMaxRelRackTop : INT ; // Max Rack in relative at the top of the Magazine
		iMaxRelRackBottom : INT ; // Max Rack in relative at the bottom of the Magazine
		
	(** PROCESS FLAG + R_Trig **)
		bButtonSettingsSave : BOOL ; // Button for save the settings of the Magazine and refresh them
			rtSettingsSave : R_Trig ; // Trigger for save the settings of the Magazine and refresh them
			
END_STRUCT
END_TYPE

// ---- 13_HMI/01_DUTs/02_ST/ST_HMI_Magazine_Teach.TcDUT
//-----------------------------------------------------------------------------------------
//
//                  			ST_HMI_Magazine_Teach
//
//				Structure datas pour le teaching des emplacements du magasin			
//-----------------------------------------------------------------------------------------
//
//Auteur: G.GOETZ
//Création: 18.03.2026
//Dernière modification : 18.03.2026 (G.GOETZ)
//       			
//-----------------------------------------------------------------------------------------
//
//     							Liste des modifications  	
//
// 18.03.2026 (G.GOETZ) -> Création		
//-----------------------------------------------------------------------------------------

TYPE ST_HMI_Magazine_Teach :
STRUCT
	
	(** PROCESS STRING **)
		sTeachLocationSelected : STRING ;  // Number of the selected Location

	(** PROCESS INT **)
		iTeachLocationSelected : INT ; // Number of the selected Location
		
	(** PROCESS FLAG + R_Trig **)
		bVisuTeachRack : BOOL ; // Schow the Teach Rack button if the selected Location is the first of them
		bVisuTeachAllTop : BOOL ; // Schow the Teach AllTop button if the selected Location is the first of them
		bVisuTeachAllBottom : BOOL ; // Schow the Teach AllBottom button if the selected Location is the first of them
	
		bButtonTeachLocation : BOOL ; // Button for teach the selected Locaiton
			rtTeachLocation : R_Trig ; // Trigger for teach the selected Locaiton
		bButtonTeachRack : BOOL ; // Button for teach the Rack of the selected Location
			rtTeachRack : R_Trig ; // Trigger for teach the Rack of the selected Location
		bButtonTeachAllTop : BOOL ; // Button for teach AllTop Locaiton
			rtTeachAllTop: R_Trig ; // Trigger for teach AllTop Locaiton	
		bButtonTeachAllBottom : BOOL ; // Button for teach AllBottom Locaiton
			rtTeachAllBottom: R_Trig ; // Trigger for teach AllBottom Locaiton	
			
END_STRUCT
END_TYPE

// ---- 13_HMI/01_DUTs/02_ST/ST_HMI_Manipulator_Gripper.TcDUT
//-----------------------------------------------------------------------------------------
//
//                  			ST_HMI_Manipulator_Gripper
//
//						Structure datas pour la pince du manipulateur 		
//-----------------------------------------------------------------------------------------
//
//Auteur: G.GOETZ
//Création: 09.02.2026
//Dernière modification : 09.02.2026 (G.GOETZ)
//       			
//-----------------------------------------------------------------------------------------
//
//     							Liste des modifications  	
//
// 09.02.2026 (G.GOETZ) -> Création		
//-----------------------------------------------------------------------------------------

TYPE ST_HMI_Manipulator_Gripper :
STRUCT

	(** SETUP TIME **)
		tMouvementOpen : TIME ; // Value of the open mouvement duration
		tMouvementClose : TIME ; // Value of the close mouvement duration
	
	(** SETUP INT **)
		iMouvementOpen : INT ; // Value of the open mouvement duration
		iMouvementClose : INT ; // Value of the close mouvement duration
	
	(** SETUP FLAG **)
		bCheckSensorOpen : BOOL ; // Check the sensor after open mouvement
		bCheckSensorClose : BOOL ; // Check the sensor after close mouvement
		
	(** PROCESS FLAG + R_TRIG **)
		bButtonOpenManupulatorGripper : BOOL ; // Button for open the gripper of the Manipulator
			rtOpenManupulatorGripper : R_Trig ; // Trigger for open the gripper of the Manipulator
		bButtonCloseManupulatorGripper : BOOL ; // Button for open the gripper of the Manipulator
			rtCloseManupulatorGripper : R_Trig ; // Trigger for open the gripper of the Manipulator
	
END_STRUCT
END_TYPE

// ---- 13_HMI/01_DUTs/02_ST/ST_HMI_Manipulator_Breakage.TcDUT
//-----------------------------------------------------------------------------------------
//
//                  			ST_HMI_Manipulator_Breakage
//
//					Structure datas pour le bris outil via le manipulateur 	
//-----------------------------------------------------------------------------------------
//
//Auteur: G.GOETZ
//Création: 06.02.2026
//Dernière modification : 06.02.2026 (G.GOETZ)
//       			
//-----------------------------------------------------------------------------------------
//
//     							Liste des modifications  	
//
// 06.02.2026 (G.GOETZ) -> Création		
//-----------------------------------------------------------------------------------------

TYPE ST_HMI_Manipulator_Breakage :
STRUCT

	(** SETUP TIME **)
		tTimeout : TIME ; // Value of the timeout for the breakage ctrl
	
	(** SETUP LREAL **)
		lrOffsetSensor : LREAL ; // Offset position above the breakage sensor
		lrToleranceLength : LREAL ; // Tolerance for tool length
		lrMeasureVelocity : LREAL ; // Velocity for the measure

	(** SETUP INT **)
		iTimeout : INT ; // Value of the timeout for the breakage ctrl
	
END_STRUCT
END_TYPE

// ---- 13_HMI/01_DUTs/02_ST/ST_HMI_Manipulator_Tunnel.TcDUT
//-----------------------------------------------------------------------------------------
//
//                  			ST_HMI_Manipulator_Tunnel
//
//				Structure datas pour le passage du tunnel du manipulateur 			
//-----------------------------------------------------------------------------------------
//
//Auteur: G.GOETZ
//Création: 06.02.2026
//Dernière modification : 06.02.2026 (G.GOETZ)
//       			
//-----------------------------------------------------------------------------------------
//
//     							Liste des modifications  	
//
// 06.02.2026 (G.GOETZ) -> Création		
//-----------------------------------------------------------------------------------------

TYPE ST_HMI_Manipulator_Tunnel :
STRUCT
	
	(** SETUP TIME **)
		tTimeout : TIME ; // Value of the timeout for travel the tunnel

	(** SETUP INT **)
		iTimeout : INT ; // Value of the timeout for travel the tunnel

END_STRUCT
END_TYPE

// ---- 13_HMI/01_DUTs/02_ST/ST_HMI_Pick_Tool_Magazine.TcDUT
//-----------------------------------------------------------------------------------------
//
//                  			ST_HMI_Pick_Tool_Magazine
//
//							Structure HMI prise outil dans magasin		
//-----------------------------------------------------------------------------------------
//
//Auteur: G.GOETZ
//Création: 20.02.2026
//Dernière modification : 20.02.2026 (G.GOETZ)
//       			
//-----------------------------------------------------------------------------------------
//
//     							Liste des modifications  	
//
// 20.02.2026 (G.GOETZ) -> Création		
//-----------------------------------------------------------------------------------------

TYPE ST_HMI_Pick_Tool_Magazine :
STRUCT

	(** SETUP FLAG **)
		(*Manipulator*)
			bCheckSensorManipulatorGripper : BOOL ; // Check the sensor of the manipulator gripper
		(*Arm*)
			//bCheckSensorArmGripper1 : BOOL ; // Check the sensor of the arm gripper 1
			//bCheckSensorArmGripper2 : BOOL ; // Check the sensor of the arm gripper 2
	
		bCheckLocation : BOOL ; // With or Without chek Tool presence in Location before pick

END_STRUCT
END_TYPE

// ---- 13_HMI/01_DUTs/02_ST/ST_HMI_Transfer_ManipulatorToArm.TcDUT
//-----------------------------------------------------------------------------------------
//
//                  		ST_HMI_Transfer_ManipulatorToArm
//
//						Structure HMI transfert manipulateur vers bras		
//-----------------------------------------------------------------------------------------
//
//Auteur: G.GOETZ
//Création: 20.02.2026
//Dernière modification : 20.02.2026 (G.GOETZ)
//       			
//-----------------------------------------------------------------------------------------
//
//     							Liste des modifications  	
//
// 20.02.2026 (G.GOETZ) -> Création		
//-----------------------------------------------------------------------------------------

TYPE ST_HMI_Transfer_ManipulatorToArm :
STRUCT

	(** SETUP FLAG **)
		(*Manipulator*)
			bCheckSensorManipulatorGripper : BOOL ; // Check the sensor of the manipulator gripper
		(*Arm*)
			bCheckSensorArmGripper1 : BOOL ; // Check the sensor of the arm gripper 1
			bCheckSensorArmGripper2 : BOOL ; // Check the sensor of the arm gripper 2

END_STRUCT
END_TYPE

// ---- 13_HMI/01_DUTs/02_ST/ST_HMI_Screen_Home.TcDUT
//-----------------------------------------------------------------------------------------
//
//                  			ST_HMI_Screen_Home
//
//							Structure datas page Home HMI 			
//-----------------------------------------------------------------------------------------
//
//Auteur: G.GOETZ
//Création: 21.01.2026
//Dernière modification : 21.01.2026 (G.GOETZ)
//       			
//-----------------------------------------------------------------------------------------
//
//     							Liste des modifications  	
//
// 21.01.2026 (G.GOETZ) -> Création		
//-----------------------------------------------------------------------------------------


TYPE ST_HMI_Screen_Home :
STRUCT

	(** SETUP INT **)
		ix1 : INT ; // ?
	
	(** SETUP FLAG **)
		bx1 : BOOL ; // ?

	(** PROCESS INT **)
		iy1 : INT ; // ?
	
	(** PROCESS FLAG **)
		by1 : BOOL ; // ?
	
END_STRUCT
END_TYPE

// ---- 13_HMI/01_DUTs/02_ST/ST_HMI_Transfer_ArmCnc.TcDUT
//-----------------------------------------------------------------------------------------
//
//                  			ST_HMI_Transfer_ArmCnc
//
//						Structure HMI transfert entre bras et cnc		
//-----------------------------------------------------------------------------------------
//
//Auteur: G.GOETZ
//Création: 20.02.2026
//Dernière modification : 20.02.2026 (G.GOETZ)
//       			
//-----------------------------------------------------------------------------------------
//
//     							Liste des modifications  	
//
// 20.02.2026 (G.GOETZ) -> Création		
//-----------------------------------------------------------------------------------------

TYPE ST_HMI_Transfer_ArmCnc :
STRUCT

	(** SETUP FLAG **)
		(*Arm*)
			bCheckSensorArmGripper1 : BOOL ; // Check the sensor of the arm gripper 1
			bCheckSensorArmGripper2 : BOOL ; // Check the sensor of the arm gripper 2

END_STRUCT
END_TYPE

// ---- 13_HMI/01_DUTs/02_ST/ST_HMI_Transfer_ArmToManipulator.TcDUT
//-----------------------------------------------------------------------------------------
//
//                  		ST_HMI_Transfer_ArmToManipulator
//
//						Structure HMI transfert bras vers manipulateur		
//-----------------------------------------------------------------------------------------
//
//Auteur: G.GOETZ
//Création: 26.02.2026
//Dernière modification : 26.02.2026 (G.GOETZ)
//       			
//-----------------------------------------------------------------------------------------
//
//     							Liste des modifications  	
//
// 26.02.2026 (G.GOETZ) -> Création		
//-----------------------------------------------------------------------------------------

TYPE ST_HMI_Transfer_ArmToManipulator :
STRUCT

	(** SETUP FLAG **)
		(*Manipulator*)
			bCheckSensorManipulatorGripper : BOOL ; // Check the sensor of the manipulator gripper
		(*Arm*)
			bCheckSensorArmGripper1 : BOOL ; // Check the sensor of the arm gripper 1
			bCheckSensorArmGripper2 : BOOL ; // Check the sensor of the arm gripper 2

END_STRUCT
END_TYPE

// ---- 14_Log/01_DUTs/01_ENUM/ENUM_Log_File_Management.TcDUT
{attribute 'qualified_only'}
{attribute 'strict'}

//-----------------------------------------------------------------------------------------
//
//                  			ENUM_Log_File_Management
//
//									Log file management 			
//-----------------------------------------------------------------------------------------
//
//Auteur: G.GOETZ (inspired by S.MANTZER)
//Création: 04.02.2026
//Dernière modification : 04.02.2026 (G.GOETZ)
//       			
//-----------------------------------------------------------------------------------------
//
//     							Liste des modifications  	
//
// 04.02.2026 (G.GOETZ) -> Création		
//-----------------------------------------------------------------------------------------

TYPE ENUM_Log_File_Management :
(
	Automatic := 1 , 
	Manual := 2 ,	
	ManualWithDelete := 3 
);
END_TYPE

// ---- 14_Log/01_DUTs/01_ENUM/ENUM_Log_Type.TcDUT
{attribute 'qualified_only'}
{attribute 'strict'}

//-----------------------------------------------------------------------------------------
//
//                  			ENUM_Log_Type
//
//									Log type 			
//-----------------------------------------------------------------------------------------
//
//Auteur: G.GOETZ (inspired by S.MANTZER)
//Création: 04.02.2026
//Dernière modification : 04.02.2026 (G.GOETZ)
//       			
//-----------------------------------------------------------------------------------------
//
//     							Liste des modifications  	
//
// 04.02.2026 (G.GOETZ) -> Création		
//-----------------------------------------------------------------------------------------

TYPE ENUM_Log_Type :
(
	WM := 1 , 
	Customer := 2 	
);
END_TYPE

// ---- 14_Log/01_DUTs/02_ST/ST_Log.TcDUT
//-----------------------------------------------------------------------------------------
//
//                  				ST_Log
//
//								Structure Log 			
//-----------------------------------------------------------------------------------------
//
//Auteur: G.GOETZ (inspired by S.MANTZER)
//Création: 04.02.2026
//Dernière modification : 04.02.2026 (G.GOETZ)
//       			
//-----------------------------------------------------------------------------------------
//
//     							Liste des modifications  	
//
// 04.02.2026 (G.GOETZ) -> Création		
//-----------------------------------------------------------------------------------------

TYPE ST_Log :
STRUCT
	
	(** STRING **)
	strLogDateTime : STRING[50] ; // Date and Time to Log
	strLogTxt : STRING[255] ; // Text to Log
	
END_STRUCT
END_TYPE

// ---- 14_Log/01_DUTs/02_ST/ST_Log_Data.TcDUT
//-----------------------------------------------------------------------------------------
//
//                  				ST_Log_Data
//
//								Structure Log Data			
//-----------------------------------------------------------------------------------------
//
//Auteur: G.GOETZ (inspired by S.MANTZER)
//Création: 04.02.2026
//Dernière modification : 04.02.2026 (G.GOETZ)
//       			
//-----------------------------------------------------------------------------------------
//
//     							Liste des modifications  	
//
// 04.02.2026 (G.GOETZ) -> Création		
//-----------------------------------------------------------------------------------------

TYPE ST_Log_Data :
STRUCT

	(** ARRAY ST **)
	aBufferLog	: ARRAY[1..GV_log.iMaxLog] OF ST_Log ; // Buffer log	
	
	(** DATE & TIME **)
	dtLastLogDateTimeNewFile : DATE_AND_TIME  ; // Date and TIME
	
	(** INT **)
	iLineIndex : INT := 1 ;
	iFileNumber : INT := 0 ;

	(** FLAG **)	
	bBufferFull : BOOL ;

END_STRUCT
END_TYPE

// ---- 02_Events/02_GVLs/GV_Events.TcGVL
{attribute 'qualified_only'}

//-----------------------------------------------------------------------------------------
//
//                  				GV_Events
//
//								Variables évènements 			
//-----------------------------------------------------------------------------------------
//
//Auteur: G.GOETZ (inspired by S.MANTZER)
//Création: 21.01.2026
//Dernière modification : 21.01.2026 (G.GOETZ)
//       			
//-----------------------------------------------------------------------------------------
//
//     							Liste des modifications  	
//
// 21.01.2026 (G.GOETZ) -> Création		
//-----------------------------------------------------------------------------------------

VAR_GLOBAL PERSISTENT
END_VAR

VAR_GLOBAL 
	
	(** ARRAY ST **) // Data for HMI
	aEventGroup	: ARRAY[1..GV_Events.iMaxEventGroup] OF ST_EVENT_GROUP ; // Event Group Structure	
	
	(** INT **)
	iEventGroupNumberAssignement : INT := 0 ;
	iEventGroupGeneralEvent : INT := 0 ; 
	iEventGroupCallEvent : INT := 0 ; 
	
END_VAR

VAR_GLOBAL CONSTANT
	
	(** CONSTANT INT **) // Data for HMI
	iMaxEventGroup : INT := 50; // Max EVENT GROUP 1-60 
	iMaxAlarms : INT := 200; // Max Alarms by EVENT GROUP	
	iMaxMessages : INT := 50; // Max Messages by EVENT GROUP			
	iMaxOpMessages : INT := 50; // Max Operator Messages by EVENT GROUP
	
END_VAR

// ---- 03_Operating_Mode/02_GVLs/GV_OpMode.TcGVL
{attribute 'qualified_only'}

//-----------------------------------------------------------------------------------------
//
//                  				GV_OpMode
//
//								Variables op Mode 			
//-----------------------------------------------------------------------------------------
//
//Auteur: G.GOETZ
//Création: 20.02.2026
//Dernière modification : 20.02.2026 (G.GOETZ)
//       			
//-----------------------------------------------------------------------------------------
//
//     							Liste des modifications  	
//
// 20.02.2026 (G.GOETZ) -> Création		
//-----------------------------------------------------------------------------------------

VAR_GLOBAL PERSISTENT
END_VAR

VAR_GLOBAL
	
	(** ENUM **)
		eOpModeRequest : ENUM_OpMode := ENUM_OpMode.None ;
		eOpMode : ENUM_OpMode := ENUM_OpMode.None ;

	(** PROCESS FLAG **)
		bInitAllowed : BOOL ; // Init is Allowed
		bAutoAllowed : BOOL ; // Auto is Allowed
		bManuAllowed : BOOL ; // Manu is Allowed

END_VAR

VAR_GLOBAL CONSTANT
END_VAR

// ---- 05_Fans/02_GVLs/GV_Fans.TcGVL
{attribute 'qualified_only'}

//-----------------------------------------------------------------------------------------
//
//                  				GV_Fans
//
//							Variables ventilateur(s) 			
//-----------------------------------------------------------------------------------------
//
//Auteur: G.GOETZ
//Création: 20.01.2026
//Dernière modification : 20.01.2026 (G.GOETZ)
//       			
//-----------------------------------------------------------------------------------------
//
//     							Liste des modifications  	
//
// 20.01.2026 (G.GOETZ) -> Création		
//-----------------------------------------------------------------------------------------

VAR_GLOBAL PERSISTENT
END_VAR

VAR_GLOBAL
	
	(** ARRAY ST **)
	aId	: ARRAY[1..iMaxFans] OF ST_Fan ; // Fan Structure
	
	(** REAL **)
	rTempArmor : REAL ; // Temp of the Electrical Armor
	rTempArmorFiltered : REAL ; // Temp Filtered of the Electrical Armor
	
	(** ST **)
	stMisc : ST_Miscellaneous ; // Miscellaneous if need
	
END_VAR

VAR_GLOBAL CONSTANT
	
	(** CONSTANT UINT **)
	uRampStep1 : UINT := 1 ; //  step ramp for the fan accel and decel

	(** CONSTANT INT **)
	iMaxFans : INT := 1 ; // Max Fans
	
END_VAR

// ---- 06_Doors/02_GVLs/GV_Doors.TcGVL
{attribute 'qualified_only'}

//-----------------------------------------------------------------------------------------
//
//                  				GV_Doors
//
//								Variables porte(s) 			
//-----------------------------------------------------------------------------------------
//
//Auteur: G.GOETZ (inspired by S.MANTZER)
//Création: 13.01.2026
//Dernière modification : 13.01.2026 (G.GOETZ)
//       			
//-----------------------------------------------------------------------------------------
//
//     							Liste des modifications  	
//
// 13.01.2026 (G.GOETZ) -> Création		
//-----------------------------------------------------------------------------------------

VAR_GLOBAL PERSISTENT
END_VAR

VAR_GLOBAL
	
	(** ARRAY ST **)
		aId	: ARRAY[1..iMaxDoors] OF ST_Door ; // Door Structure
	
	(** PROCESS FLAG **)
		bDoorsCloseLock : BOOL := FALSE ; //Doors OK
	
	(** ST **)
		stMisc : ST_Miscellaneous ; // Miscellaneous if need
	
END_VAR

VAR_GLOBAL CONSTANT
	
	(** CONSTANT INT **)
		iMaxDoors : INT := 1; // Max Doors
	
END_VAR

// ---- 07_Cyltronic/02_GVLs/CTC_CONSTANTS.TcGVL
VAR_GLOBAL
	CTC_MOTION_MODE_OFF 		:USINT := 0;
	CTC_MOTION_MODE_HALT 		:USINT := 1;
	CTC_MOTION_MODE_TEACH 		:USINT := 2;
	CTC_MOTION_MODE_MOVEOUT 	:USINT := 3;
	CTC_MOTION_MODE_MOVEIN 		:USINT := 4;
	CTC_MOTION_MODE_FREEPOS 	:USINT := 5;
	CTC_MOTION_MODE_FREEPOSPRO 	:USINT := 6;
	CTC_MOTION_MODE_HOME 		:USINT := 7;
	CTC_MOTION_MODE_RESET 		:USINT := 255;
	CTC_MOTION_MODE_FREEPOSREL 	:USINT := 30;
	CTC_MOTION_MODE_FREEVEL 	:USINT := 31;
	CTC_MOTION_MODE_FREETORQUE 	:USINT := 32;
	CTC_MOTION_MODE_DONOTHING	:USINT := 128;
	//	
	CTC_STATUS_BYTE_IDLE 		:USINT := 0;
	CTC_STATUS_BYTE_READY 		:USINT := 1;
	CTC_STATUS_BYTE_ACTIVE 		:USINT := 2;
	CTC_STATUS_BYTE_ERROR 		:USINT := 3;
	CTC_STATUS_BYTE_TEACH 		:USINT := 4;
END_VAR

// ---- 07_Cyltronic/02_GVLs/GV_Cyltronic.TcGVL
{attribute 'qualified_only'}

//-----------------------------------------------------------------------------------------
//
//                  				GV_Cyltronic
//
//								Variables Cyltronic 			
//-----------------------------------------------------------------------------------------
//
//Auteur: G.GOETZ
//Création: 04.03.2026
//Dernière modification : 04.03.2026 (G.GOETZ)
//       			
//-----------------------------------------------------------------------------------------
//
//     							Liste des modifications  	
//
// 04.03.2026 (G.GOETZ) -> Création		
//-----------------------------------------------------------------------------------------

VAR_GLOBAL PERSISTENT
END_VAR

VAR_GLOBAL
	
	(** ARRAY ST **)
		aId	: ARRAY[1..iMaxCyltronic] OF ST_Cyltronic ; // Cyltronic Structure
	
	(** PROCESS FLAG **)
	
	(** ST **)
		stMisc : ST_Miscellaneous ; // Miscellaneous if need
	
END_VAR

VAR_GLOBAL CONSTANT
	
	(** CONSTANT INT **)
		iMaxCyltronic : INT := 1 ; // Max Cyltronic
	
END_VAR

// ---- 08_Cycle/02_GVLs/GV_Cycle.TcGVL
{attribute 'qualified_only'}

//-----------------------------------------------------------------------------------------
//
//                  				GV_Cycle
//
//								Variables cycle 			
//-----------------------------------------------------------------------------------------
//
//Auteur: G.GOETZ
//Création: 02.02.2026
//Dernière modification : 02.02.2026 (G.GOETZ)
//       			
//-----------------------------------------------------------------------------------------
//
//     							Liste des modifications  	
//
// 02.02.2026 (G.GOETZ) -> Création		
//-----------------------------------------------------------------------------------------

VAR_GLOBAL PERSISTENT
	
	(** PROCESS ARRAY ENUM **)
		aSequence  : ARRAY[1..iMaxActions] OF ENUM_Cycle_Action ; // Sequence in Actions of the Cycle
	
	(** PROCESS ENUM **)
		eCycleStep : ENUM_Cycle_Step ; // Steps for the cycle
		eCyclePrevStep : ENUM_Cycle_Step ; // Previous Step of the cycle in progress
		eCycleType : ENUM_Cycle_Type ; // Type of th cycle
	
	(** PROCESS UDINT **)
		udiErrorID : UDINT ; // ErrorID Cycle
	
	(** PROCESS INT **)
		iSeqLength : INT ; // Number of Actions in the Sequence
		iSeqIndex : INT ; // Action in progress in the Sequence
		
		iArmGripperLoad : INT ; // Gripper number to load on the changing arm
		iArmGripperUnload : INT ; // Gripper number to unload on the changing arm

		iGripperArmToCncNumber : INT ; // Gripper number to transfer from changing arm to cnc spindle
		iGripperCncToArmNumber : INT ; // Gripper number to transfer from cnc spindle to changing arm
		
		iSpindleToolLocation : INT ; // Spindle Tool Location for the cycle (memory at the beggining, can't change durnig the cycle)
		iToolToLoadLocationRel : INT ; // Relative Tool To Load Location for the cycle (memory at the beggining, can't change durnig the cycle)
		iToolToLoadLocationAbs : INT ; // Absolute Tool To Load Location for the cycle (memory at the beggining, can't change durnig the cycle)
		iToolToUnloadLocationRel : INT ; // Relative Tool To UnLoad Location for the cycle (memory at the beggining, can't change durnig the cycle)
		iToolToUnloadLocationAbs : INT ; // Absolute Tool To UnLoad Location for the cycle (memory at the beggining, can't change durnig the cycle)
	
		iToolToCheckLocationAbs : INT ; // Absolute Tool To Check Location
	
	(** PROCESS FLAG **)
		bStartStop : BOOL ; // Start/Stop Cycle
		
		bInitSet : BOOL ; // fb_Init.bInit is Set
		
		bInitRequest : BOOL ; // InitRequest
		bInitCycleDone : BOOL ; // InitCycle is Done
	
		bCycleInProgress: BOOL ; // Cycle in progress
		bActionRunning : BOOL ; // Action is Running
		bActionError : BOOL ; // Action in Error
		bResetError : BOOL ; // Reset Error
		
		bAnticipateLoadRequest1 : BOOL ; // Request to anticipate the Pick Tool in Magazine
		bAnticipateLoadRequest2 : BOOL ; // Request to anticipate the Manipulator to Arm
		bAnticipateLoadDone : BOOL ; // Anticipate the Pick Tool in Magazine is Done

		bAnticipateUnloadRequest3 : BOOL ; // Request to anticipate the Arm to Manipulator
		bAnticipateUnloadRequest4 : BOOL ; // Request to anticipate the Place Tool in Magazine
		//bAnticipateUnloadDone : BOOL ; // Anticipate the Palce Tool in Magazine is Done
		
		bSpindleToolLocationCheck : BOOL ; // Check of the Spindle Tool Location Done and OK
		bToolToLoadLocationCheck : BOOL ; // Check of the Tool To Load Location Done and OK
		
		bTransferCncToArm : BOOL ; // Transfer from changing arm to cnc spindle
		bTransferArmToCnc : BOOL ; // Transfer from cnc spindle to changing arm
		
		bOpenIntermediateDoorRequest : BOOL ; // Request for open the Intermediate Door
		bCloseIntermediateDoorRequest : BOOL ; // Request for close the Intermediate Door
		
END_VAR

VAR_GLOBAL

	(** SETUP INT **)
		iEventGroup : INT := 0 ; // Group for events
		iIdHMI : INT := 0 ; // Number for events on HMI
		
	(** SETUP FLAG **)
		bEventAck : BOOL := FALSE ; // Events Acknowledgement

	(** ST **)
		stMisc : ST_Miscellaneous ; // Miscellaneous if need

END_VAR

VAR_GLOBAL CONSTANT
	
	(** CONSTANT INT **)
		iMaxActions : INT := 12 ; // Number Max of actions in a Sequence
	
END_VAR

// ---- 09_Tool_Magazine/02_GVLs/GV_Tool_Magazine.TcGVL
{attribute 'qualified_only'}

//-----------------------------------------------------------------------------------------
//
//                  				GV_Tool_Magazine
//
//								Variables magasin d'outils 			
//-----------------------------------------------------------------------------------------
//
//Auteur: G.GOETZ
//Création: 14.01.2026
//Dernière modification : 14.01.2026 (G.GOETZ)
//       			
//-----------------------------------------------------------------------------------------
//
//     							Liste des modifications  	
//
// 14.01.2026 (G.GOETZ) -> Création		
//-----------------------------------------------------------------------------------------

VAR_GLOBAL PERSISTENT

	(** ARRAY ST **)
		aLocation : ARRAY[1..iMaxAbsLocation] OF ST_Tool_Location ; // Tool_Location structure
		aCheckLocation : ARRAY[1..iMaxAbsLocation] OF ST_Tool_Location ; // Tool_Location structure for the Full Check

	(** ARRAY **)
		(* For IO/Link *)
			//aBreakageSensorIn AT %I* : ARRAY[0..1] OF BYTE ;
// 		alrXExclusionZone : ARRAY[1..10] OF LREAL ; // Exclusion Zone coordinate Axis X
// 		alrYExclusionZone : ARRAY[1..10] OF LREAL ; // Exclusion Zone coordinate Axis Y
// 		alrZExclusionZone : ARRAY[1..10] OF LREAL ; // Exclusion Zone coordinate Axis Z
// 		abExclusionZone : ARRAY[1..10] OF BOOL ; // Exclusion Zone

	(** SETUP LREAL **)  // -> from HMI st/screen : Magazine_Settings
		(* Top *)
			lrZAbsCompensationLocationTop : LREAL := 0.0 ; // Z compensation total for the locations at the top in mm
	
			lrXLocationOffsetTop : LREAL := 0.0 ; // X Offset between location at the top of the Magazine
			lrYLocationOffsetTop : LREAL := 0.0 ; // Y Offset between location at the top of the Magazine
			lrZLocationOffsetTop : LREAL := 0.0 ; // Z Offset between location at the top of the Magazine
			
			lrXFirstLocationTop : LREAL := 0.0 ; // X of the first location at the top of the Magazine (first absolute)
			lrYLocationTop : LREAL := 0.0 ; // Y of the Location at the top of the Magazine
			lrZLowestRackTop : LREAL := 0.0 ; // Z of the lowest rack at the top of the Magazine 
			
		(* Bottom *)
			lrZAbsCompensationLocationBottom : LREAL := 0.0 ; // Z compensation total for the locations at the bottom in mm
			
			lrXLocationOffsetBottom : LREAL := 0.0 ; // X Offset between location at the bottom of the Magazine
			lrYLocationOffsetBottom : LREAL := 0.0 ; // Y Offset between location at the bottom of the Magazine
			lrZLocationOffsetBottom : LREAL := 0.0 ; // Z Offset between location at the bottom of the Magazine
			
			lrXFirstLocationBottom : LREAL := 0.0 ; // X of the first location at the bottom of the Magazine (first absolute)
			lrYLocationBottom : LREAL := 0.0 ; // Y of the Location at the bottom of the Magazine
			lrZLowestRackBottom : LREAL := 0.0 ; // Z of the first lowest at the bottom of the Magazine
	
	
		lrYOffsetFrontLocation : LREAL := 0.0 ; // Y Offset to be in front of the Y coordinate of the location
		lrZOffsetAboveLocation : LREAL := 0.0 ; // Y Offset to be in front of the Y coordinate of the location

		lrZOffsetAboveArmGripper1 : LREAL := 0.0 ; // Z Offset to be above the Z coordinate of the changing arm gripper 1 when in tansfer position
		lrZOffsetAboveArmGripper2 : LREAL := 0.0 ; // Z Offset to be above the Z coordinate of the changing arm gripper 2 when in tansfer position

		lrZOffsetToolCheck : LREAL := 0.0 ; // Z Offset above the tool for the check
		lrYOffsetToolCheck : LREAL := 0.0 ; // Y Offset in front of the tool for the check

		lrZRelCompensationLocationTop : LREAL := 0.0 ; // Z compensation between each location at the top in mm
		lrZRelCompensationLocationBottom : LREAL := 0.0 ; // Z compensation between each location at the bottom in mm

	(** SETUP REAL **)
		rZBrakeTimer : REAL := 0.0 ; // Timer before brake axis Z 

	(** SETUP INT **)  // -> from HMI st/screen : Magazine_Settings
		iMaxRelRackLocationTop : INT := 0 ; // Max Location in a Rack in relative at the top of the Magazine
		iMaxRelRackLocationBottom : INT := 0 ; // Max Location in a Rack in relative at the bottom of the Magazine
		iMaxRelRackTop : INT := 0 ; // Max Rack in relative at the top of the Magazine
		iMaxRelRackBottom : INT := 0 ; // Max Rack in relative at the bottom of the Magazine

	(** SETUP INT **)
		iMaxRelLocation : INT := 0 ; // Max Location in relative in the Magazine
		iMaxRelLocationTop : INT := 0 ; // Max Location in relative at the top of the Magazine
		iMaxRelLocationBottom : INT := 0 ; // Max Location in relative at the bottom of the Magazine
		iMaxRelRack : INT := 0 ; // Max Rack in relative in the Magazine
	
	(** PROCESS LREAL **)
		lrMinXTeach : LREAL := 0.0 ;
		lrMaxXTeach : LREAL := 0.0 ;
		lrMinYTeach : LREAL := 0.0 ;
		lrMaxYTeach : LREAL := 0.0 ;
		lrMinZTeach : LREAL := 0.0 ;
		lrMaxZTeach : LREAL := 0.0 ;
		
	(** PROCESS UINT **)
	 	uiBreakageSensor AT %I* : UINT ; //Input Tool Measure sensor
	
	(** PROCESS FLAG **)
//		bExclusionZone : BOOL ; // Exclusion Zone is Activ
	
		bFirstCycleCheckMagazine : BOOL ; // Check the Magazine after First Cycle
		bCheckFullMagazineRequest : BOOL ; // Request for Full Check the Magazine
		bCheckFullMagazineDone : BOOL ; // Full Check of the Magazine is Done
		bCheckOneMagazineRequest : BOOL ; // Request for Check one Location in the Magazine
		bCheckOneMagazineDone : BOOL ; // One Location Check in the Magazine is Done
		
		bCheckManipulatorMemoryRequest : BOOL ; // Request for Check Manipulator memory in the Magazine
		bCheckArmGripper1MemoryRequest : BOOL ; // Request for Check Arm Gripper 1 memory in the Magazine
		bCheckArmGripper2MemoryRequest : BOOL ; // Request for Check Arm Gripper 2 memory in the Magazine
		bCheckSpindleMemoryRequest : BOOL ; // Request for Check Spindle memory in the Magazine
		
		bAuthorizationTeachLocation : BOOL ; // Authorization to teach the selected Location
		bAuthorizationTeachRack : BOOL ; // Authorization to teach the Rack of the selected Location
		bAuthorizationTeachAllTop : BOOL ; // Authorization to teach AllTop Location
		bAuthorizationTeachAllBottom : BOOL ; // Authorization to teach AllBottom Location

		bAuthorizationTeachPositions : BOOL ; // Authorization to teach Positions

	(** ST **)
		stManipulator : ST_Manipulator_Head ; // Manipulator_Head structure
		stArm : ST_Changing_Arm ; // Changing_Arm structure
	
END_VAR

VAR_GLOBAL

	(** SETUP INT **)
		iEventGroup : INT := 0 ; // Group for events

	(** PROCESS INT **)
		iCheckLocationTopSize : INT := 0 ; // Number of Location on the Top in the aCheckLocation Array
		iCheckLocationBottomSize : INT := 0 ; // Number of Location on the Bottom in the aCheckLocation Array
	
	(** PROCESS FLAG **)
		bFullCheckMagazineInitLocation : BOOL := FALSE ; // Start the Init of the Location data for the Check Magazine
	
	(** ST **)
		stMisc : ST_Miscellaneous ; // Miscellaneous if need	

END_VAR

VAR_GLOBAL CONSTANT
		
	(** CONSTANT LREAL **)
		lrMinAbsCompensationLocationTop : LREAL := -5.0 ; // Min Compensation in absolute for the Location at the top of the Magazine
		lrMaxAbsCompensationLocationTop : LREAL := 5.0 ; // Max Compensation in absolute for the Location at the top of the Magazine
		lrMinAbsCompensationLocationBottom : LREAL := -5.0 ; // Min Compensation in absolute for the Location at the bottom of the Magazine
		lrMaxAbsCompensationLocationBottom : LREAL := 5.0 ; // Max Compensation in absolute for the Location at the bottom of the Magazine
	
		lrMinXLocationOffsetTop : LREAL := 30.0 ; // Min X Offset between location at the top of the Magazine
		lrMaxXLocationOffsetTop : LREAL := 40.0 ; // Max X Offset between location at the top of the Magazine
		lrMinYLocationOffsetTop : LREAL := -5.0 ; // Min Y Offset between location at the top of the Magazine
		lrMaxYLocationOffsetTop : LREAL := 5.0 ; // Max Y Offset between location at the top of the Magazine
		lrMinZLocationOffsetTop : LREAL := 110.0 ; // Min Z Offset between location at the top of the Magazine
		lrMaxZLocationOffsetTop : LREAL := 130.0 ; // Max Z Offset between location at the top of the Magazine

		lrMinXLocationOffsetBottom : LREAL := 30.0 ; // Min X Offset between location at the bottom of the Magazine
		lrMaxXLocationOffsetBottom : LREAL := 40.0 ; // Max X Offset between location at the bottom of the Magazine
		lrMinYLocationOffsetBottom : LREAL := 0.0 ; // Min Y Offset between location at the bottom of the Magazine
		lrMaxYLocationOffsetBottom : LREAL := 10.0 ; // Max Y Offset between location at the bottom of the Magazine
		lrMinZLocationOffsetBottom : LREAL := 140.0 ; // Min Z Offset between location at the bottom of the Magazine
		lrMaxZLocationOffsetBottom : LREAL := 160.0 ; // Max Z Offset between location at the bottom of the Magazine
		
		lrMinYOffsetFrontLocation : LREAL := 40.0 ; // Min Y Offset to be in Front of the Location in the Magazine
		lrMaxYOffsetFrontLocation : LREAL := 60.0 ; // Max Y Offset to be in Front of the Location in the Magazine

		lrMinZOffsetAboveLocation : LREAL := 15.0 ; // Min Z Offset to be Above of the Location in the Magazine
		lrMaxZOffsetAboveLocation : LREAL := 20.0 ; // Max Z Offset to be Above of the Location in the Magazine
		
		lrMinZOffsetAboveArmGripper1 : LREAL := 15.0 ; // Min Z Offset to be Above the transfer position of the ArmGripper1
		lrMaxZOffsetAboveArmGripper1 : LREAL := 25.0 ; // Max Z Offset to be Above the transfer position of the ArmGripper1
		lrMinZOffsetAboveArmGripper2 : LREAL := 15.0 ; // Min Z Offset to be Above the transfer position of the ArmGripper2
		lrMaxZOffsetAboveArmGripper2 : LREAL := 25.0 ; // Max Z Offset to be Above the transfer position of the ArmGripper2
		
		lrMinZOffsetToolCheck : LREAL := 15.0 ; // Min Z Offset to be Above of the Location in the Magazine for the check
		lrMaxZOffsetToolCheck : LREAL := 20.0 ; // Max Z Offset to be Above of the Location in the Magazine for the check
		lrMinYOffsetToolCheck : LREAL := -10.0 ; // Min Z Offset to be Above of the Location in the Magazine for the check
		lrMaxYOffsetToolCheck : LREAL := 0.0 ; // Max Z Offset to be Above of the Location in the Magazine for the check
		
		lrMinXFirstLocationTop : LREAL := 30.0 ; // Min X of the First Location at the top of the Magazine
		lrMaxXFirstLocationTop : LREAL := 685.0 ; // Max X of the First Location at the top of the Magazine
		lrMinXFirstLocationBottom : LREAL := 170.0 ; // Min X of the First Location at the bottom of the Magazine
		lrMaxXFirstLocationBottom : LREAL := 685.0 ; // Max X of the First Location at the bottom of the Magazine
		
		lrMinYLocationTop : LREAL := 70.0 ; // Min Y of the Location at the top of the Magazine
		lrMaxYLocationTop : LREAL := 72.5 ; // Max Y of the Location at the top of the Magazine
		lrMinYLocationBottom : LREAL := 70 ; // Min Y of the Location at the bottom of the Magazine
		lrMaxYLocationBottom : LREAL := 72.5 ; // Max Y of the Location at the bottom of the Magazine
		
		lrMinZLowestRackTop : LREAL := 650 ; // Min Z of the Lowest Rack at the top of the Magazine
		lrMaxZLowestRackTop : LREAL := 1150 ; // Max Z of the Lowest Rack at the top of the Magazine
		lrMinZLowestRackBottom : LREAL := 1 ; // Min Z of the Lowest Rack at the bottom of the Magazine
		lrMaxZLowestRackBottom : LREAL := 350 ; // Max Z of the Lowest Rack at the bottom of the Magazine
		
	(** CONSTANT INT **)
		iMaxAbsRackTop : INT := 5 ; // Max Rack in absolute at the top of the Magazine
		iMaxAbsRackBottom : INT := 3 ; // Max Rack in absolute at the bottom of the Magazine
		iMaxAbsRack : INT := iMaxAbsRackTop+iMaxAbsRackBottom ; // Max Rack in absolute in the Magazine
	
		iMaxAbsLocationRackTop : INT := 19 ; // Max Location in absolute in a Rack at the top
		iMaxAbsLocationRackBottom : INT := 15 ; // Max Location in absolute in a Rack at the bottom
		
		iMaxAbsLocationTop : INT := iMaxAbsRackTop*iMaxAbsLocationRackTop ; // Max Location in absolute at the top of the Magazine
		iMaxAbsLocationBottom : INT := iMaxAbsRackBottom*iMaxAbsLocationRackBottom ; // Max Location in absolute at the bottom of the Magazine
		iMaxAbsLocation : INT := iMaxAbsLocationTop+iMaxAbsLocationBottom ; // Max Location in absolute in the Magazine
		
		//iMaxSmallDiam : INT := 30 ; // Max diameter for a small tool
		//iMaxSmallLength : INT := 60 ; // Max length of a small tool
		
		iNumCharaToolName: INT := 30 ; // Number of characters for a tool name
	
	(** CONSTANT ST **)
		stEmptyToolLocation : ST_Tool_Location ; // Empty Tool_Location structure
		stEmptyToolParam : ST_Tool_Parameters ; // Empty Tool Parameters structure
		stEmptyToolName : ST_Tool_Name ; // Empty Tool Name structure
	
END_VAR

// ---- 10_Axes/02_GVLs/GV_Axes.TcGVL
{attribute 'qualified_only'}

//-----------------------------------------------------------------------------------------
//
//                  				GV_Axes
//
//							Variables pour les Axes
//-----------------------------------------------------------------------------------------
//
//Auteur: G.GOETZ
//Création: 28.01.2026
//Dernière modification : 28.01.2026 (G.GOETZ)
//       			
//-----------------------------------------------------------------------------------------
//
//     							Liste des modifications  	
//
// 28.01.2026 (G.GOETZ) -> Création		
//-----------------------------------------------------------------------------------------

VAR_GLOBAL PERSISTENT

	(** ST **)
		stAxisX : ST_Axis ; // Structure Axis
		stAxisY : ST_Axis ; // Structure Axis
		stAxisZ : ST_Axis ; // Structure Axis
		stAxisArm : ST_Axis ; // Structure Axis

END_VAR

VAR_GLOBAL

	(** PROCESS ENUM **)
		eJogAxisSelect : ENUM_Axis_Select := ENUM_Axis_Select.None ; // Axis Selected for Jog
		eJogAxisRequest : ENUM_Axis_Select := ENUM_Axis_Select.None ; // Axis Request for Jog

		eJogDirection : ENUM_Jog_Direction := ENUM_Jog_Direction.None ; // Direction for jog
		eJogMode : ENUM_Jog_Mode := ENUM_Jog_Mode.None ; // Mode for jog	
	
		eRefAxisSelect : ENUM_Axis_Select := ENUM_Axis_Select.None ; // Axis Selected for Referencing
		eRefAxisRequest : ENUM_Axis_Select := ENUM_Axis_Select.None ; // Axis Request for Referencing

	(** PROCESS TIME **)
		tBrakeAxisZ : TIME ; // Time after a mouvement to set the brake of the Axis Z
		
	(** PROCESS LREAL **)
		lrVelocityAxisX : LREAL ; // Velocity Axis X
		lrVelocityAxisY : LREAL ; // Velocity Axis Y
		lrVelocityAxisZ : LREAL ; // Velocity Axis Z
		lrVelocityAxisArm : LREAL ; // Velocity Axis Arm
		
	(** PROCESS FLAG **)	
		//bJogRequestRisingEdge : BOOL ; // Rising Edge for Jog Request	
		bAxisAllDisabled : BOOL ; // All Axis are disabled
		bAxisAllNotMoving : BOOL ; // All Axis are not moving
		bAxisAllOperational : BOOL ; // All Axis are operational
		bAxisXAllowed : BOOL ; // Select Axis X is Allowed
		bAxisYAllowed : BOOL ; // Select Axis Y is Allowed
		bAxisZAllowed : BOOL ; // Select Axis Z is Allowed
		bAxisArmAllowed : BOOL ; // Select Axis Arm is Allowed
		
		bReferencingXAllowed : BOOL ; // Select Referencing X is Allowed
		bReferencingYAllowed : BOOL ; // Select Referencing Y is Allowed
		bReferencingZAllowed : BOOL ; // Select Referencing Z is Allowed
		bReferencingArmAllowed : BOOL ; // Select Referencing Arm is Allowed

	(** ST **)
		stMisc : ST_Miscellaneous ; // Miscellaneous if need
	
END_VAR

VAR_GLOBAL CONSTANT

	(** CONSTANT LREAL **)
		lrAutoMaxSpeedAxisX : LREAL := 697.0 ; // Max Speed in AUTO for the Axis X (mm/s)
		lrAutoMaxSpeedAxisY : LREAL := 169.0 ; // Max Speed in AUTO for the Axis Y (mm/s)
		lrAutoMaxSpeedAxisZ : LREAL := 384.0 ; // Max Speed in AUTO for the Axis Z (mm/s)
		lrAutoMaxSpeedAxisArm : LREAL := 578.0 ; // Max Speed in AUTO for the Axis Arm (mm/s)
		
		lrJogMaxSpeedAxisX : LREAL := 30 ; //lrAutoMaxSpeedAxisX/10 ; // Max Speed in Jog for the Axis X (mm/s)
		lrJogMaxSpeedAxisY : LREAL := 15 ; //lrAutoMaxSpeedAxisY/10 ; // Max Speed in Jog for the Axis Y (mm/s)
		lrJogMaxSpeedAxisZ : LREAL := 30 ; //lrAutoMaxSpeedAxisZ/10 ; // Max Speed in Jog for the Axis Z (mm/s)
		lrJogMaxSpeedAxisArm : LREAL := 30 ; //lrAutoMaxSpeedAxisArm/10 ; // Max Speed in Jog for the Axis Arm (mm/s)
	
END_VAR

// ---- 10_Axes/02_GVLs/GV_Handwheel.TcGVL
{attribute 'qualified_only'}

//-----------------------------------------------------------------------------------------
//
//                  				GV_Handwheel
//
//						Variables boitier manivelle du magasin doutils 			
//-----------------------------------------------------------------------------------------
//
//Auteur: G.GOETZ
//Création: 19.01.2026
//Dernière modification : 19.01.2026 (G.GOETZ)
//       			
//-----------------------------------------------------------------------------------------
//
//     							Liste des modifications  	
//
// 19.01.2026 (G.GOETZ) -> Création		
//-----------------------------------------------------------------------------------------

VAR_GLOBAL PERSISTENT

	(** ARRAY ST **)
		aId	: ARRAY[1..iMaxHandwheels] OF ST_Handwheel ; // Door Structure	

END_VAR

VAR_GLOBAL
	
	(** ST **)
		stMisc : ST_Miscellaneous ; // Miscellaneous if need
	
END_VAR

VAR_GLOBAL CONSTANT
	
	(** CONSTANT TIME **)
		tPowerTime : TIME := T#3S ; // Power time
		tInactivityTime : TIME := T#300S ; // Inactivity time : 300s = 5 Minutes

	(** CONSTANT LREAL **)
		lrUnitIncrx1 : LREAL := 0.001 ; // Unit of Incremental x1 (mm)
		lrUnitIncrx10 : LREAL := 0.010 ; // Unit of Incremental x1 (mm)
		lrUnitIncrx100 : LREAL := 0.100 ; // Unit of Incremental x1 (mm)
		lrUnitIncrx1000 : LREAL := 1.000 ; // Unit of Incremental x1 (mm)
		
	(** CONSTANT INT **)
		iMaxHandwheels : INT := 1; // Max Handwheels
		iPowerValue : INT := 15172 ; // Analog_output Value : 5V = 10V/2 = 32767/2 = 16383.5 (16384=5.4V -> 15172=5V (303=0.1V))
	
END_VAR

// ---- 11_CNC/02_GVLs/GV_CNC.TcGVL
{attribute 'qualified_only'}

//-----------------------------------------------------------------------------------------
//
//                  				GV_CNC
//
//								Variables CNC 			
//-----------------------------------------------------------------------------------------
//
//Auteur: G.GOETZ
//Création: 27.01.2026
//Dernière modification : 27.01.2026 (G.GOETZ)
//       			
//-----------------------------------------------------------------------------------------
//
//     							Liste des modifications  	
//
// 27.01.2026 (G.GOETZ) -> Création		
//-----------------------------------------------------------------------------------------

VAR_GLOBAL PERSISTENT

	(** ALARMS FLAG **)
		bAlLife : BOOL ; // Life bit alarm
		bAlEmergencyStop : BOOL ; // Emergency stop alarm
		bAlNoPower : BOOL ; // No Power alarm
		bAlNoAir : BOOL ; // No Air alarm
		bAlCncFault : BOOL ; // CNC in fault alarm
		bAlCommunication : BOOL ; // Communication alarm
		bAlFocas : BOOL ; // Focas Error
	
	(** SETUP ENUM **)
		eType : ENUM_CNC_Type ; // Type of the CNC
	
	(** SETUP FLAG **)
		bEventAck : BOOL := FALSE ; // Events Acknowledgement
		bPresence : BOOL := FALSE ; // CNC presence or not
		bEnable : BOOL := FALSE ; // CNC enable or not
		bFocas : BOOL := FALSE ; // With Focas or not
		
	(** PROCESS FLAG **)
	
	(** ST **)
		stSpindle : ST_Spindle ; // Spindle structure
		
		stFanucData : ST_CNC_Fanuc_Data ; // Structure CNC Fanuc data
		stHeidenhainData : ST_CNC_Heidenhain_Data ; // Structure CNC Heidenhain data	

END_VAR

VAR_GLOBAL

	(** SETUP INT **)
		iEventGroup : INT := 0 ; // Group for events
	
	(** PROCESS INT **)
		iCommunicationStatus : INT ; // Communication Status with the CNC
	
	(** PROCESS FLAG **)	
		bReady : BOOL ; // CNC is ready
	
	(** ST **)
		stMisc : ST_Miscellaneous ; // Miscellaneous if need

END_VAR

VAR_GLOBAL CONSTANT
	
END_VAR

// ---- 12_Focas/02_GVLs/GV_Focas.TcGVL
{attribute 'qualified_only'}

//-----------------------------------------------------------------------------------------
//
//                  					GV_Focas
//
//						Variables Focas (FOCAS<->C#<->PLC(ads)) 			
//-----------------------------------------------------------------------------------------
//
//Auteur: G.GOETZ
//Création: 20.01.2026
//Dernière modification : 20.01.2026 (G.GOETZ)
//       			
//-----------------------------------------------------------------------------------------
//
//     							Liste des modifications  	
//
// 20.01.2026 (G.GOETZ) -> Création		
//-----------------------------------------------------------------------------------------

VAR_GLOBAL PERSISTENT
END_VAR

VAR_GLOBAL
	
	(** ST **)
	stFocasMagazine : ST_Focas_To_Magazine ; // Exchange Focas to Magazine
	stMagazineFocas : ST_Magazine_To_Focas ; // Exchange Magazine to Focas

	stMisc : ST_Miscellaneous ; // Miscellaneous if need	

	(** STRING **)
		sErrorAds : STRING ; // ADS Error Text

	(** INT **)
		iErrorAdsID : INT ; // ADS Error ID

	(** FLAG **)
		bLifeFlag : BOOL := FALSE ; // Bit de vie envoyé par la passerelle

	(** CONNECION FOCAS **)
		(* CommFocas STRING *)
			sFocasError : STRING ; // Description du code d'erreur
			sFocasAdr : STRING ; // Adresse IPv4 de la focas
		(* CommFocas INT *)
			iFocasErrorID : INT ; // Retourne la valeur si une erreur est survenue
			iFocasPort : INT ; // Numéro de port pour la communication avec la Focas
		(* CommFocas FLAG *)
			bFocasOK : BOOL ; // Connexion à la Focas ok
			bFocasAdsOK : BOOL ; // Connexion à l'ads ok
			bFocasStartComm : BOOL ; // Start la communication Focas
			bFocasStopComm : BOOL ; // Stop la communication 
			bFocasBusy : BOOL ; // Bloc en cours d'exécution
			bFocasDone : BOOL ; // Bloc a correctement exécuter sans erreur

	(** READ FOCAS **)
		(* ReadFocas ST *)
			stRead : St_Read_Focas ; // Tableau pour permettre plusieurs Bloc Read
		(* ReadFocas STRING *)
			sReadError : STRING ; // Description du code d'erreur
		(* ReadFocas INT *)
			iReadErrorID : INT ; // Retourne la valeur si une erreur est survenue
			iReadStep : INT ; // Etape pour le cycle de lecture
		(* ReadFocas BYTE *)
			byReadFlag : BYTE := 0 ; // Numéro du bit à lire dans un byte
		(* ReadFocas FLAG *)
			bReadStart : BOOL := FALSE ; 
			bReadBusy : BOOL ; // Vrai si le bloc réalise la requête
			bReadDone : BOOL ; // Vrai si le bloc à réaliser la requête sans problème
			
	(** WRITE FOCAS **)
		(* WriteFocas ST *)
			stWrite : St_Write_Focas ; // Tableau pour permettre plusieurs Bloc Write
		(* WriteFocas STRING *)
			sWriteError : STRING ; // Description du code d'erreur
		(* WriteFocas INT *)
			iWriteErrorID : INT ; // Retourne la valeur si une erreur est survenue
			iWriteStep : INT ; // Etape pour le cycle d'écriture
		(* WriteFocas FLAG *)
			bWriteStart : BOOL := FALSE ; 
			bWriteBusy : BOOL ; // Vrai si le bloc réalise la requête
			bWriteDone : BOOL ; // Vrai si le bloc à réaliser la requête sans problème

END_VAR

VAR_GLOBAL CONSTANT
END_VAR

// ---- 13_HMI/02_GVLs/GV_HMI.TcGVL
{attribute 'qualified_only'}

//-----------------------------------------------------------------------------------------
//
//                  				GV_HMI
//
//								Variables porte(s) 			
//-----------------------------------------------------------------------------------------
//
//Auteur: G.GOETZ 
//Création: 13.01.2026
//Dernière modification : 13.01.2026 (G.GOETZ)
//       			
//-----------------------------------------------------------------------------------------
//
//     							Liste des modifications  	
//
// 13.01.2026 (G.GOETZ) -> Création
//-----------------------------------------------------------------------------------------

VAR_GLOBAL PERSISTENT

	(** STRING **)
		sCurrentUserName : STRING ; // Current user name
		sUserMessage : STRING ; // Message for the user
		
	(** INT **)
		iCurrentScreenNumber : INT ; // Number of the current screen
		iCurrentLanguage : INT ; // Current language (1=FRENCH / 2=ENGLISH / 3=GERMAN / 4=ITALIAN)
		iCurrentUserLevel : INT ; // Current user level
	
	(** FLAG **)
		bAlarm : BOOL ; // a Alarm is available
		bMessage : BOOL ; // a Message is available
		
	(** ST **)
		stMagazineSettings : ST_HMI_Magazine_Settings ; // Structure for the magazine settings
		stMagazineTeach : ST_HMI_Magazine_Teach ; // Structure for teach the magazine
		
		stLampsLights : ST_HMI_Lamps_Lights ; // Structure for lamps and lights
		stDoors : ST_HMI_Doors ; // Structure for doors
		stCyltronic : ST_HMI_Cyltronic ; // Structure for Cyltronic // Devrait etre un tableau de taille comme dans GV_Cyltronic
		stAxes : ST_HMI_Axes ; // Structure for Axes
		stCycle : ST_HMI_Cycle ; // Structure for Cycle
		stManipulatorGripper : ST_HMI_Manipulator_Gripper ; // Structure for the manipulator gripper
		stManipulatorTunnel : ST_HMI_Manipulator_Tunnel ; // Structure for the manipulator tunnel
		stManipulatorBreakage : ST_HMI_Manipulator_Breakage ; // Structure for the manipulator breakage
		
		stMagazineCheck : ST_HMI_Magazine_Check ; // Structure for the magazine check
		
		stPickToolMagazine : ST_HMI_Pick_Tool_Magazine ; // Structure for pick tool in magazine
		stTransferManipulatorToArm : ST_HMI_Transfer_ManipulatorToArm ; // Structure for transfert manipulator to arm
		stTransferArmCnc : ST_HMI_Transfer_ArmCnc ; // Structure for transfert between arm and cnc
		stTransferArmToManipulator : ST_HMI_Transfer_ArmToManipulator ; // Structure for transfert arm to manipulator
		
		stBackup : ST_HMI_Backup ; // STructure for Backup
		
END_VAR

VAR_GLOBAL

	(** STRING **)
		sSelectBackupFile : STRING ; // Name of the selected Backup File choose by the user

	(** FLAG + R_Trig **)
		bButtonEventAck : BOOL ; // Button for Events Acknowledgement
			rtEventAck : R_Trig ; // Trigger for Events Acknowledgement
		bEventAck : BOOL ; // Events Acknowledgement

		bButtonINIT : BOOL ; // Button INIT
			rtINIT : R_Trig ; // Trigger for INIT
		bButtonAUTO : BOOL ; // Button AUTO
			rtAUTO : R_Trig ; // Trigger for AUTO
		bButtonMANU : BOOL ; // Button MANU
			rtMANU : R_Trig ; // Trigger for MANU
			
		bButtonHandwheelEnable : BOOL ; // Button for enable the Handwheel
			rtHandwheelEnable : R_Trig ; // Trigger for enable the Handwheel
			bStateHandwheelEnable : BOOL ; // State button for enable the Handwheel

		bButtonHandwheelIncr : BOOL ; // Button for handwhell in Incr mode
			rtHandwheelIncr : R_Trig ; // Trigger for handwhell in Incr mode
		bButtonHandwheelJog : BOOL ; // Button for handwhell in Jog mode
			rtHandwheelJog : R_Trig ; // Trigger for handwhell in Jog mode
		bStateHandwheelMode : BOOL ; // State of the Handwheel mode
			
		bEnableResetManipulatorMemory : BOOL ; // Enable to reset the Manipulator memory
		bEnableResetArmGripper1Memory : BOOL ; // Enable to reset the Changing Arm Gripper 1 memory
		bEnableResetArmGripper2Memory : BOOL ; // Enable to reset the Changing Arm Gripper 2 memory
		bEnableResetSpindleMemory : BOOL ; // Enable to reset the CNC Spindle memory

		bButtonRefreshToolMagazine : BOOL ; // Button for refresh the tool Magazine
			rtRefreshToolMagazine : R_Trig ; // Trigger for refresh the tool Magazine
		bButtonResetDataManipulator : BOOL ; // Button for reset the Mnipulator Head data
			rtResetDataManipulator : R_Trig ; // Trigger for reset the Mnipulator Head data
		bButtonResetDataChangingGripper1 : BOOL ; // Button for reset the Gripper 1 data of the Changing Arm
			rtResetDataChangingGripper1 : R_Trig ; // Trigger for reset the Gripper 1 data of the Changing Arm
		bButtonResetDataChangingGripper2 : BOOL ; // Button for reset the Gripper 2 data of the Changing Arm
			rtResetDataChangingGripper2 : R_Trig ; // Trigger for reset the Gripper 2 data of the Changing Arm
		bButtonResetDataSpindle : BOOL ; // Button for reset the Spindle data in CNC
			rtResetDataSpindle : R_Trig ; // Trigger for reset the Spindle data in CNC

		bButtonCncEnable : BOOL ; // Button for enable CNC
			rtCncEnable : R_TRIG ; // Trigger for enable CNC
			bStateCncEnable : BOOL ; // State button for enable CNC

		bButtonReboot : BOOL ; // Button for reboot the Magazine PC
			rtReboot : R_Trig ; // Trigger for reboot the Magazine PC
		bButtonShutdown : BOOL ; // Button for shutdown the Magazine PC
			rtShutdown : R_Trig ; // Trigger for shutdown the Magazine PC
			
	(** ST **)
		stMisc : ST_Miscellaneous ; // Miscellaneous if need	
		
END_VAR

VAR_GLOBAL CONSTANT
	
	(** CONSTANT INT **)
		iMaxScreenNumber : INT := 999 ; // Max Screen Number
	
END_VAR

// ---- 14_Log/02_GVLs/GV_Log.TcGVL
{attribute 'qualified_only'}

//-----------------------------------------------------------------------------------------
//
//                  				GV_Log
//
//								Variables Log 			
//-----------------------------------------------------------------------------------------
//
//Auteur: G.GOETZ (inspired by S.MANTZER)
//Création: 04.02.2026
//Dernière modification : 04.02.2026 (G.GOETZ)
//       			
//-----------------------------------------------------------------------------------------
//
//     							Liste des modifications  	
//
// 04.02.2026 (G.GOETZ) -> Création		
//-----------------------------------------------------------------------------------------

VAR_GLOBAL PERSISTENT

	(** ARRAY R_TRIG **)
	aLogTrig : ARRAY [1..250] OF R_TRIG;	

	(** ST **)
	stLogWM : ST_Log_Data ; // WM Log
	stLogCustom : ST_Log_Data ; // Custom Log
	
END_VAR

VAR_GLOBAL
	
	(** ST **)
	stMisc : ST_Miscellaneous ; // Miscellaneous if need
	
END_VAR

VAR_GLOBAL CONSTANT
	
	(** CONSTANT INT **)
	iMaxLog : INT := 100; // Max Log Line into buffer
	iMaxLogFile : INT := 100; // Max Log file
	
END_VAR

// ---- 02_Events/03_POUs/02_FBs/FB_Event_Group_Number_Assignement.TcPOU
FUNCTION_BLOCK FB_Event_Group_Number_Assignement
VAR_INPUT
END_VAR
VAR_OUTPUT
END_VAR
VAR
END_VAR
VAR_IN_OUT
	(** INT **)
	iEventGroup : INT ; // Number of event group
END_VAR

//-----------------------------------------------------------------------------------------
//
//                  	FB_Event_Group_Number_Assignement
//
//				Gestion assignement numéro de groupe d'évènements   			
//-----------------------------------------------------------------------------------------
//
//Auteur: G.GOETZ (inspired by S.MANTZER)
//Création: 21.01.2026
//Dernière modification : 21.01.2026 (G.GOETZ)
//       			
//-----------------------------------------------------------------------------------------
//
//     							Liste des modifications  	
//
// 21.01.2026 (G.GOETZ) -> Création		
//-----------------------------------------------------------------------------------------

(** Automatic event group number assignement **)
	IF GV_General.bFirstCycleTask THEN
		iEventGroup:=0;
		iEventGroup:=GV_Events.iEventGroupNumberAssignement;
		GV_Events.iEventGroupNumberAssignement:=GV_Events.iEventGroupNumberAssignement+1;
	ELSE
		IF iEventGroup=0 THEN
			iEventGroup:=GV_Events.iEventGroupNumberAssignement;
			GV_Events.iEventGroupNumberAssignement:=GV_Events.iEventGroupNumberAssignement+1;
		END_IF
	END_IF

END_FUNCTION_BLOCK

// ---- 02_Events/03_POUs/02_FBs/FB_Event_HMI.TcPOU
FUNCTION_BLOCK FB_Event_HMI
VAR_INPUT
	(** STRING **)	
	strEventType : STRING[20] ; // Type of the Event (ALARM or MESSAGE)
	
	(** INT **)
	iEventGroup : INT ; // Event group number
	iIdEvent : INT ; // Event Number

	(** FLAG **)
	bEventSet : BOOL ; // True to set the Event
END_VAR
VAR_OUTPUT
END_VAR
VAR
	(** FLAG **)
	bError : BOOL ; // Error
END_VAR

//-----------------------------------------------------------------------------------------
//
//                  			FB_Event_HMI
//
//						Gestion évènements pour HMI  			
//-----------------------------------------------------------------------------------------
//
//Auteur: G.GOETZ (inspired by S.MANTZER)
//Création: 21.01.2026
//Dernière modification : 21.01.2026 (G.GOETZ)
//       			
//-----------------------------------------------------------------------------------------
//
//     							Liste des modifications  	
//
// 21.01.2026 (G.GOETZ) -> Création		
//-----------------------------------------------------------------------------------------

(* Initialized variables *)
	bError:=FALSE;

(* Check EVENT GROUP, ID event, EVENT TYPE *)
	IF (iEventGroup<=0 OR iEventGroup>GV_Events.iMaxEventGroup) THEN
		GV_Events.aEventGroup[GV_Events.iEventGroupCallEvent].aMessage[5].fbMessage.Send(0); // Set Message 5 (FB_EVENT EVENT GROUP number error)
		bError:=TRUE;
	ELSE
		IF  (strEventType<>'ALARM' AND strEventType<>'MESSAGE' AND strEventType<>'OpMESSAGE') THEN
			GV_Events.aEventGroup[GV_Events.iEventGroupCallEvent].aMessage[4].fbMessage.Send(0); // Set Message 4 (FB_EVENT Event type error)
			bError:=TRUE;
		ELSE
			IF ((iIdEvent<=0 OR iIdEvent>GV_Events.iMaxAlarms) AND strEventType='ALARM') THEN
				GV_Events.aEventGroup[GV_Events.iEventGroupCallEvent].aMessage[2].fbMessage.Send(0); // Set Message 2 (FB_EVENT Alarm number error)
				bError:=TRUE;
			END_IF
			IF ((iIdEvent<=0 OR iIdEvent>GV_Events.iMaxMessages) AND strEventType='MESSAGE') THEN
				GV_Events.aEventGroup[GV_Events.iEventGroupCallEvent].aMessage[3].fbMessage.Send(0); // Set Message 3 (FB_EVENT Message number error)
				bError:=TRUE;
			END_IF	
			IF ((iIdEvent<=0 OR iIdEvent>GV_Events.iMaxOPMessages) AND strEventType='OpMESSAGE') THEN
				GV_Events.aEventGroup[GV_Events.iEventGroupCallEvent].aMessage[6].fbMessage.Send(0); // Set Message 6 (FB_EVENT Operator Message number error)
				bError:=TRUE;
			END_IF		
		END_IF
	END_IF

